BC00520=86202,981627,1075175
BC00521=81835,980250,1075175
BC00522=86350,984014,1075175
BC00523=118186,882849,1075175
BC00524=118313,879045,1075175
BC00525=118363,877523,1075175
BC00526=127351,877496,1075175
BC00527=127300,879018,1075175
BC00528=127173,882822,1075175
BC00529=149531,895732,1075175
BC00530=148249,891267,1075175
BC00531=148034,889482,1075175
BC00532=151775,889498,1075175
BC00533=152288,891284,1075175
BC00534=153569,895750,1075175
BC00535=119302,902119,1075175
BC00536=119440,897649,1075175
BC00537=119495,895861,1075175
BC00538=115974,895890,1075175
BC00539=115919,897678,1075175
BC00540=115781,902148,1075175
BC00541=206850,915693,1075175
BC00542=246637,921611,1075175
BC00543=251241,924622,1075175
BC00544=253082,925827,1075175
BC00545=305626,902567,1075175
BC00546=289523,905356,1075175
BC00547=289523,905356,1075175
BC00548=265997,901694,1075172
BC00549=265782,900020,1075175
BC00550=265246,895833,1075175
BC00551=152805,918674,1075175
BC00552=155644,922700,1075175
BC00553=156780,924310,1075175
BC00554=187141,913105,1075175
BC00555=135499,922155,1075175
BC00556=202417,924491,1075175
BC00557=204603,922909,1075175
BC00558=210067,918954,1075175
BC00559=285493,836258,1075175
BC00560=322674,778579,1075175
BC00561=322674,778579,1075175
BC00562=322674,778579,1075175
BC00563=322674,778579,1075175
BC00564=322674,778579,1075175
BC00565=322674,778579,1075175
BC00566=322674,778579,1075175
BC00567=322674,778579,1075175
BC00568=272555,769164,1075175
BC00569=266479,768023,1075175
BC00570=266479,768023,1075175
BC00571=267479,770239,1071365
BC00572=266799,769335,1075175
BC00573=266479,768023,1075175
BC00574=266479,768023,1075175
BC00575=266479,768023,1075175
BC00576=266479,768023,1075175
BC00577=235984,786404,1075175
BC00578=235984,786404,1075175
BC00579=235984,786404,1075175
BC00580=235984,786404,1075175
BC00581=235984,786404,1075175
BC00582=235984,786404,1075175
BC00583=235984,786404,1075175
BC00584=235984,786404,1075175
BC00585=237203,787368,1075175
BC00586=295022,827394,1075175
BC00587=205701,931185,1075175
BC00588=204812,932218,1075175
BC00589=205671,937629,1075175
BC00590=206015,939793,1075175
BC00591=202546,941762,1075175
BC00592=218293,952795,1075175
BC00593=218466,950486,1075175
BC00594=218898,944716,1075175
BC00595=188226,925402,1075175
BC00596=189298,932104,1075175
BC00597=189728,934784,1075175
BC00598=185375,937227,1075175
BC00599=184946,934546,1075175
BC00600=183874,927845,1075175
BC00601=163256,940528,1075175
BC00602=166760,944877,1075175
BC00603=168161,946617,1075175
BC00604=172960,943924,1075175
BC00605=171559,942185,1075175
BC00606=168055,937836,1075175
BC00607=205604,952176,1075175
BC00608=237375,964309,1075175
BC00609=234858,970014,1075175
BC00610=233851,972296,1075175
BC00611=237408,970622,1075175
BC00612=238426,968449,1075175
BC00613=241139,962660,1075175
BC00614=186195,958850,1075175
BC00615=137530,955476,1075175
BC00616=142340,959691,1075175
BC00617=135217,966057,1075175
BC00618=135217,966057,1075175
BC00619=134381,966543,1075175
BC00620=132263,964948,1075175
BC00621=126968,960962,1075175
BC00622=137530,955476,1075175
BC00623=284870,850327,1075175
BC00624=323104,941595,1075175
BC00625=324436,944989,1075175
BC00626=324969,946346,1075175
BC00627=379859,936839,1075175
BC00628=379326,935482,1075175
BC00629=377994,932088,1075175
BC00630=387025,925803,1075175
BC00631=391871,922431,1075175
BC00632=387133,926188,1075175
BC00633=385238,927691,1075175
BC00634=381091,925537,1075175
BC00635=365308,912570,1075175
BC00636=363166,908743,1075175
BC00637=364796,906869,1075175
BC00638=368870,902183,1075175
BC00639=358157,902408,1075175
BC00640=354876,908652,1075175
BC00641=353564,911150,1075175
BC00642=349138,907302,1075175
BC00643=357572,916934,1075175
BC00644=359178,914754,1075175
BC00645=363193,909304,1075175
BC00646=322758,853588,1075175
BC00647=135439,955204,1075175
BC00648=139952,957848,1075175
BC00649=141757,958906,1075175
BC00650=133040,997822,1075175
BC00651=133065,977483,1075175
BC00652=144047,1040883,1075175
BC00653=142698,1043050,1075175
BC00654=139327,1048468,1075175
BC00655=142698,1043050,1075175
BC00656=21214,672831,1075175
BC00657=48829,688840,1075175
BC00658=366911,902233,1075175
BC00659=366911,902233,1075175
BC00660=366911,902233,1075175
BC00661=366911,902233,1075175
BC00662=366911,902233,1075175
BC00663=366911,902233,1075175
BC00664=366911,902233,1075175
BC00665=366911,902233,1075175
BC00666=333056,895412,1075175
BC00667=333056,895412,1075175
BC00668=333056,895412,1075175
BC00669=333056,895412,1075175
BC00670=333056,895412,1075175
BC00671=333056,895412,1075175
BC00672=333056,895412,1075175
BC00673=333056,895412,1075175
BC00674=358091,902222,1075175
BC00675=358091,902222,1075175
BC00676=358091,902222,1075175
BC00677=358091,902222,1075175
BC00678=358091,902222,1075175
BC00679=358091,902222,1075175
BC00680=358091,902222,1075175
BC00681=358091,902222,1075175
BC00682=358091,902222,1075175
BC00683=358091,902222,1075175
BC00684=358091,902222,1075175
BC00685=358091,902222,1075175
BC00686=358091,902222,1075175
BC00687=358091,902222,1075175
BC00688=398174,894103,1075175
BC00689=398174,894103,1075175
BC00690=398174,894103,1075175
BC00691=398174,894103,1075175
BC00692=398174,894103,1075175
BC00693=398174,894103,1075175
BC00694=398174,894103,1075175
BC00695=398174,894103,1075175
BC00696=264903,781270,1075175
BC00697=264903,781270,1075175
BC00698=264904,781269,1075172
BC00699=264904,781269,1075171
BC00700=264904,781269,1075171
BC00701=264904,781269,1075168
BC00702=264904,781269,1075168
BC00703=264904,781269,1075168
BC00704=264904,781269,1075168
BC00705=264904,781269,1075168
BC00706=264904,781269,1075164
BC00707=264903,781270,1075175
BC00708=301264,775814,1075175
BC00709=301264,775814,1075175
BC00710=301264,775814,1075175
BC00711=301264,775814,1075175
BC00712=301264,775814,1075175
BC00713=301264,775814,1075175
BC00714=301264,775814,1075175
BC00715=301264,775814,1075175
BC00716=301264,775814,1075175
BC00717=301264,775814,1075175
BC00718=274235,786209,1075175
BC00719=238672,799885,1075175
BC00720=238672,799885,1075175
BC00721=238672,799885,1075175
BC00722=238672,799885,1075175
BC00723=238672,799885,1075175
BC00724=238672,799885,1075175
BC00725=238672,799885,1075175
BC00726=238672,799885,1075175
BC00727=238672,799884,1075171
BC00728=238672,799884,1075171
BC00729=238672,799885,1075175
BC00730=238672,799885,1075175
BC00731=238672,799885,1075175
BC00732=238672,799885,1075175
BC00733=318263,750454,1075175
BC00734=318263,750454,1075175
BC00735=318263,750454,1075175
BC00736=318263,750454,1075175
BC00737=318263,750454,1075175
BC00738=318263,750454,1075175
BC00739=318263,750454,1075175
BC00740=318263,750454,1075175
BC00741=318263,750454,1075175
BC00742=318263,750454,1075175
BC00743=318263,750454,1075175
BC00744=318263,750454,1075175
BC00745=318263,750454,1075175
BC00746=318263,750454,1075175
BC00747=318263,750454,1075175
BC00748=318263,750454,1075175
BC00749=318263,750454,1075175
BC00750=318263,750454,1075175
BC00751=318263,750454,1075175
BC00752=318263,750454,1075175
BC00753=318263,750454,1075175
BC00754=318263,750454,1075175
BC00755=318263,750454,1075175
BC00756=318263,750454,1075175
BC00757=318263,750454,1075175
BC00758=377114,750454,1075175
BC00759=397814,750454,1075175
BC00760=397814,750454,1075175
BC00761=397814,750454,1075175
BC00762=397814,750454,1075175
BC00763=397814,750454,1075175
BC00764=397814,750454,1075175
BC00765=397814,750454,1075175
BC00766=397814,750454,1075175
BC00767=397814,750454,1075175
BC00768=397814,750454,1075175
BC00769=397814,750454,1075175
BC00770=397814,750454,1075175
BC00771=397814,750454,1075175
BC00772=397814,750454,1075175
BC00773=397814,750454,1075175
BC00774=397814,750454,1075175
BC00775=397814,750454,1075175
BC00776=397814,750454,1075175
BC00777=397814,750454,1075175
BC00778=397814,750454,1075175
BC00779=383090,762961,1075175
BC00780=372387,772052,1075175
BC00781=296274,836703,1075175
BC00782=296274,836703,1075175
BC00783=296274,836703,1075175
BC00784=296274,836703,1075175
BC00785=296274,836703,1075175
BC00786=296274,836703,1075175
BC00787=296274,836703,1075175
BC00788=296274,836703,1075175
BC00789=296274,836703,1075175
BC00790=296274,836703,1075175
BC00791=296274,836703,1075175
BC00792=296274,836703,1075175
BC00793=296274,836703,1075175
BC00794=312215,899988,1075175
BC00795=312215,944285,1075175
BC00796=312215,944285,1075175
BC00797=312215,944285,1075175
BC00798=312215,944285,1075175
BC00799=312215,944285,1075175
BC00800=312215,944285,1075175
BC00801=312215,944285,1075175
BC00802=312215,944285,1075175
BC00803=312215,944285,1075175
BC00804=312215,944285,1075175
BC00805=312215,944285,1075175
BC00806=259299,938961,1075175
BC00807=259299,938961,1075175
BC00808=259299,938961,1075175
BC00809=259299,938961,1075175
BC00810=259299,938961,1075175
BC00811=259299,938961,1075175
BC00812=259299,938961,1075175
BC00813=259299,938961,1075175
BC00814=259299,938961,1075175
BC00815=259299,938961,1075175
BC00816=259299,938961,1075175
BC00817=259299,938961,1075175
BC00818=211531,951911,1075175
BC00819=211531,951911,1075175
BC00820=211531,951911,1075175
BC00821=211531,951911,1075175
BC00822=211531,951911,1075175
BC00823=211531,951911,1075175
BC00824=211531,951911,1075175
BC00825=211531,951911,1075175
BC00826=211531,951911,1075175
BC00827=211531,951911,1075175
BC00828=211531,951911,1075175
BC00829=182503,951872,1075175
BC00830=184369,953383,1075175
BC00831=184369,953399,1075175
BC00832=184333,953526,1075175
BC00833=184897,956550,1075175
BC00834=184333,953526,1075175
BC00835=184751,953664,1075175
BC00836=187887,953121,1075175
BC00837=184751,953664,1075175
BC00838=178222,948378,1075175
BC00839=171711,951911,1075175
BC00840=171711,959591,1075175
BC00841=171711,959591,1075175
BC00842=171711,959591,1075175
BC00843=171711,959591,1075175
BC00844=171711,959591,1075175
BC00845=171711,959591,1075175
BC00846=171711,959591,1075175
BC00847=171711,959591,1075175
BC00848=171711,959591,1075175
BC00849=182815,952263,1075175
BC00850=183711,957103,1075175
BC00851=184069,959047,1075174
BC00852=184070,959056,1075175
BC00853=184189,959079,1075175
BC00854=184752,962103,1075175
BC00855=184189,959079,1075175
BC00856=182935,952303,1075175
BC00857=182935,952303,1075175
BC00858=182935,952303,1075175
BC00859=123088,1061215,1075175
BC00860=126332,1055781,1075175
BC00861=127630,1053613,1075175
BC00862=127630,1053623,1075175
BC00863=127630,1053607,1075175
BC00864=153753,1064749,1075175
BC00865=152152,1062093,1075175
BC00866=153753,1064749,1075175
BC00867=104366,1038154,1075175
BC00868=107120,1036610,1075175
BC00869=104366,1038154,1075175
BC00870=97490,1044180,1075175
BC00871=121157,1044973,1075175
BC00872=140343,1045718,1075175
BC00873=158643,1046375,1075175
BC00874=155464,1041036,1075175
BC00875=155106,1040455,1075175
BC00876=155106,1040463,1075175
BC00877=155288,1040367,1075175
BC00878=153687,1037711,1075175
BC00879=155288,1040367,1075175
BC00880=158891,1046297,1075175
BC00881=211337,993614,1075175
BC00882=274623,983932,1075175
BC00883=371761,1043051,1075175
BC00884=331941,1063020,1075175
BC00885=331941,1063020,1075175
BC00886=331941,1063020,1075175
BC00887=331941,1063020,1075175
BC00888=331941,1063020,1075175
BC00889=331941,1063020,1075175
BC00890=331941,1063020,1075175
BC00891=331941,1063020,1075175
BC00892=331941,1063020,1075175
BC00893=331941,1063020,1075175
BC00894=331941,1063020,1075175
BC00895=331941,1063020,1075175
BC00896=331941,1063020,1075175
BC00897=371761,1043051,1075175
BC00898=371761,1043051,1075175
BC00899=371761,1043051,1075175
BC00900=371761,1043051,1075175
BC00901=371761,1043051,1075175
BC00902=371761,1043051,1075175
BC00903=371761,1043051,1075175
BC00904=371761,1043051,1075175
BC00905=371761,1043051,1075175
BC00906=371761,1043051,1075175
BC00907=371761,1043051,1075175
BC00908=371761,1043051,1075175
BC00909=371761,1043051,1075175
BC00910=371761,1043051,1075175
BC00911=371761,1043051,1075175
BC00912=314185,938855,1075175
BC00913=247671,970611,1075175
BC00914=247671,970611,1075175
BC00915=247671,970611,1075175
BC00916=247671,970611,1075175
BC00917=247671,970611,1075175
BC00918=247671,970611,1075175
BC00919=247671,970611,1075175
BC00920=247671,970611,1075175
BC00921=247671,970611,1075175
BC00922=247671,970611,1075175
BC00923=247671,970611,1075175
BC00924=247671,970611,1075175
BC00925=303037,872055,1075175
BC00926=380992,820655,1075175
BC00927=380992,820655,1075175
BC00928=380992,820655,1075175
BC00929=380992,820655,1075175
BC00930=380992,820655,1075175
BC00931=380992,820655,1075175
BC00932=380992,820655,1075175
BC00933=380992,820655,1075175
BC00934=380992,820655,1075175
BC00935=380992,820655,1075175
BC00936=380992,820655,1075175
BC00937=380992,820655,1075175
BC00938=275256,812324,1075175
BC00939=125716,897903,1075175
BC00940=125716,897903,1075175
BC00941=125716,897903,1075175
BC00942=125716,897903,1075175
BC00943=125716,897903,1075175
BC00944=125716,897903,1075174
BC00945=125716,897903,1075171
BC00946=125716,897903,1075175
BC00947=125716,897903,1075175
BC00948=125716,897903,1075175
BC00949=125716,897903,1075175
BC00950=125716,897903,1075175
BC00951=125716,897903,1075175
BC00952=325019,822543,1075229
BC00953=325019,822543,1075229
BC00954=325019,822543,1075229
BC00955=325019,822543,1075229
BC00956=325019,822543,1075229
BC00957=325019,822543,1075229
BC00958=325019,822543,1075229
BC00959=325019,822543,1075229
BC00960=325019,822543,1075229
BC00961=325019,822543,1075229
BC00962=325019,822543,1075229
BC00963=325019,822543,1075229
BC00964=240667,871930,1075210
BC00965=81335,965219,1075175
BC00966=81335,965219,1075175
BC00967=81335,965219,1075175
BC00968=81335,965219,1075175
BC00969=81335,965219,1075175
BC00970=81335,965219,1075175
BC00971=81335,965219,1075175
BC00972=81335,965219,1075175
BC00973=39891,972466,1075175
BC00974=39891,972466,1075175
BC00975=39891,972466,1075175
BC00976=39891,972466,1075175
BC00977=39891,972466,1075175
BC00978=39891,972466,1075175
BC00979=39891,972466,1075175
BC00980=39891,1005107,1075175
BC00981=39891,1005107,1075175
BC00982=39891,1005107,1075175
BC00983=39891,1005107,1075175
BC00984=39891,1005107,1075175
BC00985=39891,1005107,1075175
BC00986=39891,972466,1075175
BC00987=126064,942124,1075175
BC00988=145718,951183,1075175
BC00989=145718,951183,1075175
BC00990=145718,951183,1075175
BC00991=145718,951183,1075175
BC00992=145718,951183,1075175
BC00993=145718,951183,1075175
BC00994=145718,951183,1075175
BC00995=145718,951183,1075175
BC00996=145718,951183,1075175
BC00997=145718,951183,1075175
BC00998=145718,951183,1075175
BC00999=145718,951183,1075175
BC01000=127193,914007,1075175
BC01001=75497,867475,1075175
BC01002=75497,867475,1075175
BC01003=75497,867475,1075175
BC01004=75497,867475,1075175
BC01005=75497,867475,1075175
BC01006=75497,867475,1075175
BC01007=75497,867475,1075175
BC01008=75497,867475,1075175
BC01009=75497,867475,1075175
BC01010=75497,867475,1075175
BC01011=75497,867475,1075175
BC01012=75497,867475,1075175
BC01013=75497,867475,1075175
BC01014=75497,867475,1075175
BC01015=75497,867475,1075175
BC01016=75497,867475,1075175
BC01017=75497,867475,1075175
BC01018=58830,852413,1075175
BC01019=43274,838354,1075175
BC01020=43274,838354,1075175
BC01021=43274,838354,1075175
BC01022=43274,838354,1075175
BC01023=43274,838354,1075175
BC01024=43274,838354,1075175
BC01025=43274,838354,1075175
BC01026=43274,838354,1075175
BC01027=43274,838354,1075175
BC01028=191439,896290,1075175
BC01029=209593,874493,1075175
BC01030=209593,874493,1075175
BC01031=209593,874493,1075174
BC01032=209593,874493,1075171
BC01033=209593,874493,1075175
BC01034=209593,874493,1075175
BC01035=209216,850926,1075175
BC01036=226866,854473,1075175
BC01037=228835,855864,1075175
BC01038=228835,855864,1075175
BC01039=228834,855864,1075173
BC01040=228834,855864,1075173
BC01041=228835,855864,1075175
BC01042=228835,855864,1075175
BC01043=228835,855864,1075175
BC01044=228835,855864,1075175
BC01045=228835,855864,1075175
BC01046=212683,986357,1075175
BC01047=212683,1004517,1075175
BC01048=212247,999872,1075175
BC01049=212146,998778,1075171
BC01050=214955,996593,1075174
BC01051=222186,994128,1075175
BC01052=222622,998773,1075175
BC01053=293477,973063,1075175
BC01054=293477,973063,1075175
BC01055=293477,973063,1075175
BC01056=293477,973063,1075175
BC01057=293477,973063,1075175
BC01058=293477,973063,1075175
BC01059=293477,973063,1075175
BC01060=293477,973063,1075175
BC01061=248777,974412,1075175
BC01062=147624,1017934,1075175
BC01063=124950,1033375,1075175
BC01064=124950,1033375,1075175
BC01065=124950,1033375,1075175
BC01066=124950,1033375,1075174
BC01067=124950,1033375,1075175
BC01068=124950,1033375,1075175
BC01069=106678,1046165,1075175
BC01070=106678,1046165,1075175
BC01071=106678,1046165,1075175
BC01072=106678,1046165,1075175
BC01073=106678,1046165,1075175
BC01074=106678,1046165,1075175
BC01075=172863,1024486,1075175
BC01076=172427,1019841,1075175
BC01077=172326,1018747,1075171
BC01078=175135,1016562,1075174
BC01079=182366,1014097,1075175
BC01080=182802,1018742,1075175
BC01081=253657,993032,1075175
BC01082=253657,993032,1075175
BC01083=253657,993032,1075175
BC01084=253657,993032,1075175
BC01085=253657,993032,1075175
BC01086=253657,993032,1075175
BC01087=253657,993032,1075175
BC01088=253657,993032,1075175
BC01089=208957,994381,1075175
BC01090=107804,1037903,1075175
BC01091=85130,1053344,1075175
BC01092=85130,1053344,1075175
BC01093=85130,1053344,1075175
BC01094=85130,1053344,1075175
BC01095=85130,1053344,1075175
BC01096=85130,1053344,1075175
BC01097=66858,1066134,1075175
BC01098=66858,1066134,1075175
BC01099=66858,1066134,1075175
BC01100=66858,1066134,1075175
BC01101=66858,1066134,1075175
BC01102=66858,1066134,1075175
BC01103=106678,1034404,1075175
BC01104=288363,951317,1075175
BC01105=319880,932288,1075175
BC01106=316203,930177,1075175
BC01107=314732,929332,1075175
BC01108=314732,929332,1075175
BC01109=294141,940882,1075175
BC01110=285351,949486,1075175
BC01111=280844,953897,1075175
BC01112=254356,968931,1075172
BC01113=253996,970793,1075175
BC01114=256777,973747,1075175
BC01115=224914,994659,1075175
BC01116=193407,1014756,1075175
BC01117=196552,1009267,1075175
BC01118=197065,1008372,1075175
BC01119=197397,1007797,1075175
BC01120=196552,1009278,1075175
BC01121=193407,1014766,1075175
BC01122=170876,1031134,1075175
BC01123=153007,1044116,1075175
BC01124=153007,1044116,1075175
BC01125=155599,1038213,1075175
BC01126=156636,1035851,1075175
BC01127=230598,1025728,1075175
BC01128=222023,1030515,1075175
BC01129=222023,1030515,1075175
BC01130=118655,1062836,1075175
BC01131=118655,1062836,1075175
BC01132=118655,1062836,1075175
BC01133=176896,1055708,1075175
BC01134=225377,1010635,1075175
BC01135=228184,1010601,1075175
BC01136=235201,1010515,1075175
BC01137=242597,980334,1075175
BC01138=282680,816770,1075175
BC01139=287393,774165,1075175
BC01140=293866,776192,1075175
BC01141=296455,777002,1075175
BC01142=296337,777088,1075175
BC01143=296308,777110,1075175
BC01144=296189,777197,1075175
BC01145=293600,776386,1075175
BC01146=287127,774359,1075175
BC01147=265173,805126,1075175
BC01148=271841,806848,1075175
BC01149=274508,807537,1075175
BC01150=274508,807537,1075175
BC01151=271842,806893,1075175
BC01152=265174,805171,1075175
BC01153=347775,809657,1075175
BC01154=348436,809459,1075175
BC01155=348700,809380,1075175
BC01156=352833,807067,1075175
BC01157=364813,800347,1075175
BC01158=368942,798027,1075175
BC01159=368677,798106,1075175
BC01160=368016,798304,1075175
BC01161=368016,798304,1075175
BC01162=391344,687000,1075175
BC01163=391344,687000,1075175
BC01164=391344,687000,1075175
BC01165=391344,687000,1075175
BC01166=391344,687000,1075175
BC01167=391344,687000,1075175
BC01168=391344,687000,1075175
BC01169=391344,687000,1075175
BC01170=391344,687000,1075175
BC01171=391344,687000,1075175
BC01172=391344,687000,1075175
BC01173=391344,687000,1075175
BC01174=358873,687000,1075175
BC01175=250171,896024,1075175
BC01176=255370,893912,1075175
BC01177=257449,893067,1075174
BC01178=259851,897051,1075175
BC01179=270502,914711,1075175
BC01180=268422,915555,1075175
BC01181=263223,917668,1075175
BC01182=251695,824506,1075175
BC01183=253916,829548,1075175
BC01184=254804,831565,1075175
BC01185=231448,844598,1075175
BC01186=231448,844598,1075175
BC01187=189878,862044,1075175
BC01188=188570,860127,1075175
BC01189=185301,855336,1075175
BC01190=261332,833542,1075175
BC01191=297112,823286,1075175
BC01192=293523,829343,1075175
BC01193=292087,831765,1075175
BC01194=292088,831788,1075175
BC01195=293523,829365,1075175
BC01196=297112,823308,1075175
BC01197=297112,823286,1075175
BC01198=112345,954746,1075175
BC01199=112345,954746,1075175
BC01200=111546,959512,1075175
BC01201=111226,961418,1075175
BC01202=111226,961418,1075175
BC01203=111226,961418,1075175
BC01204=63698,969650,1075175
BC01205=63700,969637,1075175
BC01206=63700,969637,1075175
BC01207=63700,969637,1075175
BC01208=64817,962978,1075175
BC01209=55529,859309,1075175
BC01210=51595,858048,1075175
BC01211=50021,857544,1075175
BC01212=45895,833192,1075175
BC01213=46071,849801,1075175
BC01214=43912,844296,1075175
BC01215=45475,843733,1075175
BC01216=45475,843733,1075175
BC01217=45475,843733,1075175
BC01218=45475,843733,1075175
BC01219=45475,843733,1075175
BC01220=49382,842326,1075175
BC01221=32191,855540,1075175
BC01222=35199,856902,1075175
BC01223=36402,857447,1075175
BC01224=24170,872455,1075175
BC01225=24116,855865,1075175
BC01226=17601,856883,1075175
BC01227=10106,858388,1075175
BC01228=7107,859694,1075175
BC01229=124165,958731,1075175
BC01230=124477,964204,1075175
BC01231=124602,966393,1075175
BC01232=119899,967208,1075175
BC01233=114659,968116,1075175
BC01234=114534,965927,1075175
BC01235=114222,960453,1075175
BC01236=169497,963360,1075175
BC01237=218455,965934,1075175
BC01238=214431,967961,1075175
BC01239=212822,968772,1075175
BC01240=212822,968772,1075175
BC01241=212822,968772,1075175
BC01242=212822,968772,1075175
BC01243=218344,963319,1075175
BC01244=222368,961291,1075175
BC01245=147324,958268,1075175
BC01246=86350,984014,1075175
BC01247=90717,985390,1075175
BC01248=92241,985755,1075175
BC01249=87949,982178,1075175
BC01250=87949,982178,1075175
BC01251=87949,982178,1075175
BC01252=86202,981627,1075175
BC01253=81835,980250,1075175
BC01254=83182,969192,1075175
BC01255=84657,971884,1075175
BC01256=84782,974073,1075175
BC01257=80079,974888,1075175
BC01258=74839,975796,1075175
BC01259=74714,973607,1075175
BC01260=74402,968133,1075175
BC01261=129677,971040,1075175
BC01262=178635,973614,1075175
BC01263=174611,975641,1075175
BC01264=173002,976452,1075175
BC01265=173002,976452,1075175
BC01266=173002,976452,1075175
BC01267=173002,976452,1075175
BC01268=178524,970999,1075175
BC01269=182548,968971,1075175
BC01270=107504,965948,1075175
BC01271=46530,991694,1075175
BC01272=50897,993070,1075175
BC01273=52421,993435,1075175
BC01274=48129,989858,1075175
BC01275=48129,989858,1075175
BC01276=48129,989858,1075175
BC01277=46382,989307,1075175
BC01278=42015,987930,1075175
BC01279=86350,984014,1075175
BC01280=118186,882849,1075175
BC01281=118313,879045,1075175
BC01282=118363,877523,1075175
BC01283=127351,877496,1075175
BC01284=127300,879018,1075175
BC01285=127173,882822,1075175
BC01286=149531,895732,1075175
BC01287=148249,891267,1075175
BC01288=148034,889482,1075175
BC01289=151775,889498,1075175
BC01290=152288,891284,1075175
BC01291=153569,895750,1075175
BC01292=119302,902119,1075175
BC01293=119440,897649,1075175
BC01294=119495,895861,1075175
BC01295=115974,895890,1075175
BC01296=115919,897678,1075175
BC01297=115781,902148,1075175
BC01298=206850,915693,1075175
BC01299=246637,921611,1075175
BC01300=251241,924622,1075175
BC01301=253082,925827,1075175
BC01302=305626,902567,1075175
BC01303=289523,905356,1075175
BC01304=289523,905356,1075175
BC01305=265997,901694,1075172
BC01306=265782,900020,1075175
BC01307=265246,895833,1075175
BC01308=152805,918674,1075175
BC01309=155644,922700,1075175
BC01310=156780,924310,1075175
BC01311=187141,913105,1075175
BC01312=179441,914454,1075175
BC01313=179441,914454,1075175
BC01314=179441,914454,1075175
BC01315=120688,931609,1075175
BC01316=120688,931609,1036122
BC01317=120688,931609,1036122
BC01318=135499,922155,1075175
BC01319=196755,924293,1075175
BC01320=204603,922909,1075175
BC01321=210067,918954,1075175
BC01322=285493,836258,1075175
BC01323=322674,778579,1075175
BC01324=322674,778579,1075175
BC01325=322674,778579,1075175
BC01326=322674,778579,1075175
BC01327=322674,778579,1075175
BC01328=322674,778579,1075175
BC01329=322674,778579,1075175
BC01330=322674,778579,1075175
BC01331=272555,769164,1075175
BC01332=266479,768023,1075175
BC01333=266479,768023,1075175
BC01334=267479,770239,1071365
BC01335=266799,769335,1075175
BC01336=266479,768023,1075175
BC01337=266479,768023,1075175
BC01338=266479,768023,1075175
BC01339=266479,768023,1075175
BC01340=235984,786404,1075175
BC01341=235984,786404,1075175
BC01342=235984,786404,1075175
BC01343=235984,786404,1075175
BC01344=235984,786404,1075175
BC01345=235984,786404,1075175
BC01346=235984,786404,1075175
BC01347=235984,786404,1075175
BC01348=237203,787368,1075175
BC01349=295022,827394,1075175
BC01350=205701,931185,1075175
BC01351=204812,932218,1075175
BC01352=205671,937629,1075175
BC01353=206015,939793,1075175
BC01354=202546,941762,1075175
BC01355=218293,952795,1075175
BC01356=218466,950486,1075175
BC01357=218898,944716,1075175
BC01358=188226,925402,1075175
BC01359=189298,932104,1075175
BC01360=189728,934784,1075175
BC01361=185375,937227,1075175
BC01362=184946,934546,1075175
BC01363=183874,927845,1075175
BC01364=163256,940528,1075175
BC01365=166760,944877,1075175
BC01366=168161,946617,1075175
BC01367=172960,943924,1075175
BC01368=171559,942185,1075175
BC01369=168055,937836,1075175
BC01370=205604,952176,1075175
BC01371=237375,964309,1075175
BC01372=234858,970014,1075175
BC01373=233851,972296,1075175
BC01374=237408,970622,1075175
BC01375=238426,968449,1075175
BC01376=241139,962660,1075175
BC01377=186195,958850,1075175
BC01378=137530,955476,1075175
BC01379=142340,959691,1075175
BC01380=135217,966057,1075175
BC01381=135217,966057,1075175
BC01382=134381,966543,1075175
BC01383=132263,964948,1075175
BC01384=126968,960962,1075175
BC01385=137530,955476,1075175
BC01386=284870,850327,1075175
BC01387=323104,941595,1075175
BC01388=323297,942087,1075175
BC01389=323297,942087,1075175
BC01390=323297,942087,1075175
BC01391=324969,946346,1075175
BC01392=377020,937331,1075175
BC01393=379859,936839,1075175
BC01394=379326,935482,1075175
BC01395=377994,932088,1075175
BC01396=387025,925803,1075175
BC01397=391871,922431,1075175
BC01398=387133,926188,1075175
BC01399=385238,927691,1075175
BC01400=381091,925537,1075175
BC01401=365308,912570,1075175
BC01402=363166,908743,1075175
BC01403=364796,906869,1075175
BC01404=368870,902183,1075175
BC01405=358157,902408,1075175
BC01406=354876,908652,1075175
BC01407=353564,911150,1075175
BC01408=349138,907302,1075175
BC01409=357572,916934,1075175
BC01410=359178,914754,1075175
BC01411=363193,909304,1075175
BC01412=322758,853588,1075175
BC01413=135439,955204,1075175
BC01414=139952,957848,1075175
BC01415=141757,958906,1075175
BC01416=133040,997822,1075175
BC01417=133065,977483,1075175
BC01418=144047,1040883,1075175
BC01419=142698,1043050,1075175
BC01420=139327,1048468,1075175
BC01421=139327,1048468,1075175
BC01422=95619,955204,1075175
BC01423=100132,965528,1075175
BC01424=101937,966586,1075175
BC01425=93220,1005502,1075175
BC01426=93220,1005502,1075175
BC01427=93221,1030527,1075216
BC01428=93221,1030527,1075216
BC01429=99566,1045795,1075190
BC01430=142698,1043050,1075175
BC01431=206177,1018673,1075175
BC01432=252443,1048931,1075175
BC01433=258757,1029159,1075175
BC01434=290253,930536,1075175
BC01435=290253,930536,1075175
BC01436=290253,930536,1075175
BC01437=297151,966120,1075172
BC01438=297151,997903,1075172
BC01439=297151,997903,1075172
BC01440=297194,1021413,1075172
BC01441=297194,1021413,1075172
BC01442=21214,672831,1075175
BC01443=21214,672831,429902
BC01444=66815,724118,419761
BC01445=110240,772957,337669
BC01446=124996,789553,122283
BC01447=124996,789553,122283
BC01448=124996,789553,122283
BC01449=124996,789553,122283
BC01450=124996,789553,122283
BC01451=124996,789553,122283
BC01452=124996,789553,122283
BC01453=124996,789553,122283
BC01454=124996,789553,122283
BC01455=124996,789553,122283
BC01456=124996,789553,122283
BC01457=124996,789553,122283
BC01458=124996,789553,122283
BC01459=124996,789553,122283
BC01460=124996,789553,122283
BC01461=136729,789553,283981
BC01462=136729,789553,283981
BC01463=136729,789553,283981
BC01464=136729,789553,283981
BC01465=136729,789553,283981
BC01466=136729,789553,283981
BC01467=136729,789553,283981
BC01468=136729,789553,283981
BC01469=136729,789553,283981
BC01470=136729,789553,283981
BC01471=163194,789553,386705
BC01472=163194,789553,386705
BC01473=163194,789553,386705
BC01474=163194,789553,386705
BC01475=163194,789553,386705
BC01476=163194,789553,386705
BC01477=163194,789553,386705
BC01478=163194,789553,386705
BC01479=163194,789553,386705
BC01480=163194,789553,386705
BC01481=110240,772957,337669
BC01482=66815,724118,419761
BC01483=66815,670858,419761
BC01484=252765,670858,277331
BC01485=322808,760288,131711
BC01486=322808,760288,131711
BC01487=322808,760288,131711
BC01488=322808,760288,131711
BC01489=322808,760288,131711
BC01490=322808,760288,131711
BC01491=322808,760288,131711
BC01492=322808,760288,131711
BC01493=322808,760288,131711
BC01494=335534,789553,204922
BC01495=335534,789553,204922
BC01496=335534,789553,204922
BC01497=335534,789553,204922
BC01498=335534,789553,204922
BC01499=335534,789553,204922
BC01500=335534,789553,204922
BC01501=335534,789553,204922
BC01502=335534,789553,204922
BC01503=335534,789553,204922
BC01504=335534,789553,204922
BC01505=335534,789553,204922
BC01506=335534,789553,204922
BC01507=335534,789553,204922
BC01508=335534,789553,204922
BC01509=335534,789553,204922
BC01510=344006,752651,139062
BC01511=344006,752651,139062
BC01512=344005,752652,139060
BC01513=344005,752652,139060
BC01514=344005,752652,139060
BC01515=344005,752652,139060
BC01516=344005,752652,139060
BC01517=344005,752652,139060
BC01518=344005,752652,139060
BC01519=344005,752652,139060
BC01520=344005,752652,139060
BC01521=344005,752652,139060
BC01522=344005,752652,139060
BC01523=344005,752652,139060
BC01524=344005,752652,139060
BC01525=344006,752651,139062
BC01526=300933,750795,218908
BC01527=283893,750061,250495
BC01528=276320,749735,264534
BC01529=276320,749735,264534
BC01530=276320,749735,264534
BC01531=276320,749735,264532
BC01532=276320,749735,264532
BC01533=276320,749735,264532
BC01534=276320,749735,264532
BC01535=276320,749735,264532
BC01536=276320,749735,264532
BC01537=276320,749735,264532
BC01538=276320,749735,264532
BC01539=276320,749736,264531
BC01540=276320,749736,264531
BC01541=276320,749736,264531
BC01542=276320,749736,264531
BC01543=276320,749735,264534
BC01544=248857,763770,138691
BC01545=248857,763770,138691
BC01546=248857,763770,138691
BC01547=248857,763770,138691
BC01548=248857,763770,138691
BC01549=248857,763770,138691
BC01550=248857,763770,138691
BC01551=248857,763770,138691
BC01552=248857,763770,138691
BC01553=248857,763770,138691
BC01554=248857,763770,138691
BC01555=248857,763770,138691
BC01556=248857,763770,138691
BC01557=248857,763770,138691
BC01558=248857,763770,138691
BC01559=248857,763770,138691
BC01560=287864,789553,132710
BC01561=287864,789553,132710
BC01562=287864,789553,132710
BC01563=287864,789553,132710
BC01564=287864,789553,132710
BC01565=287864,789553,132710
BC01566=287864,789553,132710
BC01567=287864,789553,132710
BC01568=287864,789553,132710
BC01569=287864,789553,132710
BC01570=287864,789553,132710
BC01571=287864,789553,132710
BC01572=279829,789553,53
BC01573=279829,789553,53
BC01574=279829,789553,53
BC01575=279829,789553,53
BC01576=279829,789553,53
BC01577=279829,789553,53
BC01578=279829,789553,53
BC01579=279829,789553,53
BC01580=279829,789553,53
BC01581=279829,789553,53
BC01582=279829,789553,53
BC01583=279829,789553,53
BC01584=279829,789553,53
BC01585=312324,789553,158805
BC01586=312324,789553,158805
BC01587=312324,789553,158804
BC01588=312324,789553,158805
BC01589=312324,789553,158805
BC01590=312324,789553,158805
BC01591=303082,768394,105099
BC01592=303082,768394,105099
BC01593=303082,768394,105099
BC01594=303082,768394,105099
BC01595=303082,768394,105099
BC01596=303082,768394,105099
BC01597=287868,781442,183325
BC01598=278410,789553,231953
BC01599=278410,789553,231953
BC01600=278410,789553,231953
BC01601=278410,789553,231953
BC01602=278410,789553,231953
BC01603=278410,789553,231953
BC01604=283893,750061,250495
BC01605=300933,750795,218908
BC01606=376723,772526,120737
BC01607=376723,772526,120737
BC01608=376723,772526,120737
BC01609=376723,772526,120737
BC01610=376723,772526,120737
BC01611=376723,772526,120737
BC01612=385013,737075,95404
BC01613=385013,737075,95404
BC01614=385013,737075,95404
BC01615=385013,737075,95404
BC01616=385013,737075,95404
BC01617=385013,737075,95404
BC01618=365962,760163,122379
BC01619=365962,760163,122379
BC01620=365962,760163,122379
BC01621=365962,760163,122379
BC01622=365962,760163,122379
BC01623=365962,760163,122379
BC01624=365962,760163,122379
BC01625=252765,670858,277331
BC01626=66815,670858,419761
BC01627=66815,724118,419761
BC01628=110240,772957,337669
BC01629=118803,789553,240458
BC01630=118803,789553,240458
BC01631=118803,789553,240458
BC01632=118803,789553,240458
BC01633=118803,789553,240458
BC01634=118803,789553,240458
BC01635=130259,789553,198376
BC01636=110709,789553,198376
BC01637=113251,789553,198376
BC01638=113251,789553,198376
BC01639=113251,789553,198376
BC01640=113251,789553,198376
BC01641=113251,789553,198376
BC01642=113251,789553,198376
BC01643=113251,789553,198376
BC01644=113251,789553,198376
BC01645=113251,789553,198376
BC01646=113251,789553,198376
BC01647=113251,789553,198376
BC01648=113251,789553,198376
BC01649=113251,789553,198376
BC01650=113251,789553,228042
BC01651=113251,789553,280292
BC01652=113251,789553,280290
BC01653=113251,789553,280290
BC01654=113251,789553,280290
BC01655=113251,789553,280290
BC01656=113251,789553,280290
BC01657=113251,789553,280290
BC01658=113251,789553,280290
BC01659=110240,772957,337669
BC01660=66815,724118,419761
BC01661=66815,670858,419761
BC01662=252765,670858,277331
BC01663=298333,782774,240815
BC01664=298333,782774,240815
BC01665=298333,782774,240815
BC01666=298333,782774,240815
BC01667=298333,782774,240815
BC01668=298333,782774,240815
BC01669=277596,773081,190929
BC01670=277596,773081,190929
BC01671=277596,773081,190929
BC01672=277596,773081,190929
BC01673=277596,773081,190929
BC01674=277596,773081,190929
BC01675=252765,670858,277331
BC01676=66815,670858,419761
BC01677=66815,724118,419761
BC01678=110240,772957,337669
BC01679=116545,789553,319269
BC01680=116545,789553,319269
BC01681=116545,789553,319269
BC01682=116545,789553,319269
BC01683=116545,789553,319269
BC01684=116545,789553,319269
BC01685=104258,789553,379308
BC01686=104258,789553,379308
BC01687=104258,789553,379308
BC01688=104258,789553,379308
BC01689=104258,789553,379308
BC01690=104258,789553,379308
BC01691=110240,772957,337669
BC01692=66815,724118,419761
BC01693=66815,670858,419761
BC01694=252765,670858,277331
BC01695=286674,787255,240962
BC01696=286675,787255,240962
BC01697=286675,787255,240962
BC01698=286675,787255,240962
BC01699=286674,787255,240962
BC01700=286674,787255,240962
BC01701=267109,758037,158941
BC01702=267109,758037,158941
BC01703=267109,758037,158941
BC01704=267109,758037,158941
BC01705=267109,758037,158941
BC01706=267109,758037,158941
BC01707=283893,750061,250495
BC01708=360336,760725,110934
BC01709=360336,760725,110934
BC01710=360336,760725,110934
BC01711=360336,760725,110934
BC01712=360336,760725,110934
BC01713=360336,760725,110934
BC01714=371149,789553,191296
BC01715=371149,789553,191296
BC01716=371149,789553,191296
BC01717=371149,789553,191296
BC01718=371149,789553,191296
BC01719=371149,789553,191296
BC01720=283893,750061,250495
BC01721=292970,789553,136523
BC01722=292970,789553,136523
BC01723=292970,789553,136523
BC01724=292970,789553,136523
BC01725=292970,789553,136523
BC01726=292970,789552,136519
BC01727=292970,789553,136523
BC01728=292970,789553,136523
BC01729=256495,759418,21571
BC01730=256495,759418,21571
BC01731=256495,759418,21571
BC01732=256495,759418,21571
BC01733=256495,759418,21571
BC01734=256495,759418,21571
BC01735=256075,748610,41729
BC01736=255916,738170,60084
BC01737=255916,738170,60084
BC01738=255916,738170,60084
BC01739=255916,738170,60084
BC01740=255916,738170,60084
BC01741=255916,738170,60084
BC01742=262339,748900,193466
BC01743=165820,667836,534036
BC01744=21214,672831,1075175
EC00000=798156,1112951
EC00001=798156,1112951
EC00002=798156,1112951
EC00003=798156,1112951
EC00004=798156,1112951
EC00005=798156,1112951
EC00006=798156,1112951
EC00007=798156,1112951
EC00008=798156,1112951
EC00009=798156,1112951
EC00010=798156,1112951
EC00011=798156,1112951
EC00012=798156,1112951
EC00013=798156,1112951
EC00014=798156,1112951
EC00015=798156,1112951
EC00016=798156,1112951
EC00017=798156,1112951
EC00018=798156,1112951
EC00019=798156,1112951
EC00020=798156,1112951
EC00021=798156,1112951
EC00022=798156,1112951
EC00023=798156,1112951
EC00024=798156,1112951
EC00025=798156,1112951
EC00026=798156,1112951
EC00027=798156,1112951
EC00028=798156,1112951
EC00029=798156,1112951
EC00030=798156,1112951
EC00031=798156,1112951
EC00032=798156,1112951
EC00033=798156,1112951
EC00034=798156,1112951
EC00035=798155,1112950
EC00036=798155,1112950
EC00037=798155,1112950
EC00038=798154,1112949
EC00039=798154,1112949
EC00040=798154,1112949
EC00041=798154,1112949
EC00042=798154,1112949
EC00043=798153,1112949
EC00044=798156,1112951
EC00045=798156,1112951
EC00046=798156,1112951
EC00047=798156,1112951
EC00048=798156,1112951
EC00049=798156,1112951
EC00050=798156,1112951
EC00051=798156,1112951
EC00052=798156,1112951
EC00053=798156,1112951
EC00054=798156,1112951
EC00055=798156,1112951
EC00056=798156,1112951
EC00057=798156,1112951
EC00058=798156,1112951
EC00059=798156,1112951
EC00060=798156,1112951
EC00061=798156,1112951
EC00062=798156,1112951
EC00063=798156,1112951
EC00064=798155,1112950
EC00065=798155,1112950
EC00066=798156,1112951
EC00067=798156,1112951
EC00068=798156,1112951
EC00069=798156,1112951
EC00070=798156,1112951
EC00071=798156,1112951
EC00072=798156,1112951
EC00073=798156,1112951
EC00074=798156,1112951
EC00075=798156,1112951
EC00076=798156,1112951
EC00077=798156,1112951
EC00078=798156,1112951
EC00079=798156,1112951
EC00080=798156,1112951
EC00081=798156,1112951
EC00082=798156,1112951
EC00083=798156,1112951
EC00084=798156,1112951
EC00085=798156,1112951
EC00086=798156,1112951
EC00087=798156,1112951
EC00088=798156,1112951
EC00089=798156,1112951
EC00090=798156,1112951
EC00091=798156,1112951
EC00092=798156,1112951
EC00093=798156,1112951
EC00094=798156,1112951
EC00095=798156,1112951
EC00096=798156,1112951
EC00097=798156,1112951
EC00098=798156,1112951
EC00099=798156,1112951
EC00100=798156,1112951
EC00101=798156,1112951
EC00102=798156,1112951
EC00103=798156,1112951
EC00104=798156,1112951
EC00105=798156,1112951
EC00106=798156,1112951
EC00107=798156,1112951
EC00108=798156,1112951
EC00109=798156,1112951
EC00110=798156,1112951
EC00111=798156,1112951
EC00112=798156,1112951
EC00113=798156,1112951
EC00114=798156,1112951
EC00115=798156,1112951
EC00116=798156,1112951
EC00117=798156,1112951
EC00118=798156,1112951
EC00119=798156,1112951
EC00120=798156,1112951
EC00121=798156,1112951
EC00122=798156,1112951
EC00123=798156,1112951
EC00124=798156,1112951
EC00125=798156,1112951
EC00126=798156,1112951
EC00127=798156,1112951
EC00128=798156,1112951
EC00129=798156,1112951
EC00130=798156,1112951
EC00131=798156,1112951
EC00132=798156,1112951
EC00133=798156,1112951
EC00134=798156,1112951
EC00135=798156,1112951
EC00136=798156,1112951
EC00137=798156,1112951
EC00138=798156,1112951
EC00139=798156,1112951
EC00140=798156,1112951
EC00141=798156,1112951
EC00142=798156,1112951
EC00143=798156,1112951
EC00144=798156,1112951
EC00145=798156,1112951
EC00146=798156,1112951
EC00147=798156,1112951
EC00148=798156,1112951
EC00149=798156,1112951
EC00150=798156,1112951
EC00151=798156,1112951
EC00152=798156,1112951
EC00153=798156,1112951
EC00154=798156,1112951
EC00155=798156,1112951
EC00156=798156,1112951
EC00157=798156,1112951
EC00158=798156,1112951
EC00159=798156,1112951
EC00160=798156,1112951
EC00161=798156,1112951
EC00162=798156,1112951
EC00163=798156,1112951
EC00164=798156,1112951
EC00165=798156,1112951
EC00166=798156,1112951
EC00167=798156,1112951
EC00168=798156,1112951
EC00169=798156,1112951
EC00170=798156,1112951
EC00171=798156,1112951
EC00172=798156,1112951
EC00173=798156,1112951
EC00174=798156,1112951
EC00175=798156,1112951
EC00176=798156,1112951
EC00177=798156,1112951
EC00178=798155,1112950
EC00179=798156,1112951
EC00180=798156,1112951
EC00181=798156,1112951
EC00182=798156,1112951
EC00183=798156,1112951
EC00184=798156,1112951
EC00185=798156,1112951
EC00186=798156,1112951
EC00187=798156,1112951
EC00188=798156,1112951
EC00189=798156,1112951
EC00190=798156,1112951
EC00191=798156,1112951
EC00192=798156,1112951
EC00193=798156,1112951
EC00194=798156,1112951
EC00195=798156,1112951
EC00196=798156,1112951
EC00197=798156,1112951
EC00198=798156,1112951
EC00199=798156,1112951
EC00200=798156,1112951
EC00201=798156,1112951
EC00202=798156,1112951
EC00203=798156,1112951
EC00204=798156,1112951
EC00205=798156,1112951
EC00206=798156,1112951
EC00207=798156,1112951
EC00208=798156,1112951
EC00209=798156,1112951
EC00210=798156,1112951
EC00211=798156,1112951
EC00212=798156,1112951
EC00213=798156,1112951
EC00214=798156,1112951
EC00215=798156,1112951
EC00216=798156,1112951
EC00217=798156,1112951
EC00218=798156,1112951
EC00219=798156,1112951
EC00220=798156,1112951
EC00221=798156,1112951
EC00222=798156,1112951
EC00223=798156,1112951
EC00224=798156,1112951
EC00225=798156,1112951
EC00226=798156,1112951
EC00227=798156,1112951
EC00228=798156,1112951
EC00229=798156,1112951
EC00230=798156,1112951
EC00231=798156,1112951
EC00232=798156,1112951
EC00233=798156,1112951
EC00234=798156,1112951
EC00235=798156,1112951
EC00236=798156,1112951
EC00237=798156,1112951
EC00238=798156,1112951
EC00239=798156,1112951
EC00240=798156,1112951
EC00241=798156,1112951
EC00242=798156,1112951
EC00243=798156,1112951
EC00244=798156,1112951
EC00245=798156,1112951
EC00246=798156,1112951
EC00247=798156,1112951
EC00248=798156,1112951
EC00249=798156,1112951
EC00250=798156,1112951
EC00251=798156,1112951
EC00252=798156,1112951
EC00253=798156,1112951
EC00254=798156,1112951
EC00255=798156,1112951
EC00256=798155,1112951
EC00257=798156,1112951
EC00258=798156,1112951
EC00259=798156,1112951
EC00260=798156,1112951
EC00261=798156,1112951
EC00262=798156,1112951
EC00263=798156,1112951
EC00264=798156,1112951
EC00265=798156,1112951
EC00266=798156,1112951
EC00267=798156,1112951
EC00268=798156,1112951
EC00269=798156,1112951
EC00270=798156,1112951
EC00271=798156,1112951
EC00272=798156,1112951
EC00273=798156,1112951
EC00274=798156,1112951
EC00275=798156,1112951
EC00276=798156,1112951
EC00277=798156,1112951
EC00278=798156,1112951
EC00279=798156,1112951
EC00280=798156,1112951
EC00281=798156,1112951
EC00282=798156,1112951
EC00283=798156,1112951
EC00284=798156,1112951
EC00285=798156,1112951
EC00286=798156,1112951
EC00287=798156,1112951
EC00288=798156,1112951
EC00289=798156,1112951
EC00290=798156,1112951
EC00291=798156,1112951
EC00292=798156,1112951
EC00293=798156,1112951
EC00294=798156,1112951
EC00295=798156,1112951
EC00296=798156,1112951
EC00297=798156,1112951
EC00298=798156,1112951
EC00299=798156,1112951
EC00300=798156,1112951
EC00301=798156,1112951
EC00302=798156,1112951
EC00303=798156,1112951
EC00304=798156,1112951
EC00305=798156,1112951
EC00306=798156,1112951
EC00307=798156,1112951
EC00308=798156,1112951
EC00309=798156,1112951
EC00310=798156,1112951
EC00311=798156,1112951
EC00312=798156,1112951
EC00313=798156,1112951
EC00314=798156,1112951
EC00315=798156,1112951
EC00316=798156,1112951
EC00317=798156,1112951
EC00318=798156,1112951
EC00319=798156,1112951
EC00320=798156,1112951
EC00321=798156,1112951
EC00322=798156,1112951
EC00323=798156,1112951
EC00324=798156,1112951
EC00325=798156,1112951
EC00326=798156,1112951
EC00327=798156,1112951
EC00328=798156,1112951
EC00329=798156,1112951
EC00330=798156,1112951
EC00331=798156,1112951
EC00332=798156,1112951
EC00333=798156,1112951
EC00334=798156,1112951
EC00335=798156,1112951
EC00336=798156,1112951
EC00337=798155,1112950
EC00338=798156,1112951
EC00339=798156,1112951
EC00340=798156,1112951
EC00341=798156,1112951
EC00342=798156,1112951
EC00343=798156,1112951
EC00344=798155,1112951
EC00345=798155,1112951
EC00346=798156,1112951
EC00347=798156,1112951
EC00348=798156,1112951
EC00349=798156,1112951
EC00350=798156,1112951
EC00351=798156,1112951
EC00352=798156,1112951
EC00353=798156,1112951
EC00354=798155,1112950
EC00355=798156,1112951
EC00356=798156,1112951
EC00357=798156,1112951
EC00358=798156,1112951
EC00359=798156,1112951
EC00360=798156,1112951
EC00361=798156,1112951
EC00362=798156,1112951
EC00363=798156,1112951
EC00364=798156,1112951
EC00365=798156,1112951
EC00366=798156,1112951
EC00367=798156,1112951
EC00368=798156,1112951
EC00369=798156,1112951
EC00370=798156,1112951
EC00371=798156,1112951
EC00372=798156,1112951
EC00373=798156,1112951
EC00374=798156,1112951
EC00375=798156,1112951
EC00376=798156,1112951
EC00377=798156,1112951
EC00378=798156,1112951
EC00379=798156,1112951
EC00380=798156,1112951
EC00381=798156,1112951
EC00382=798156,1112951
EC00383=798156,1112951
EC00384=798156,1112951
EC00385=798156,1112951
EC00386=798156,1112951
EC00387=798156,1112951
EC00388=798156,1112951
EC00389=798155,1112950
EC00390=798156,1112951
EC00391=798156,1112951
EC00392=798156,1112951
EC00393=798156,1112951
EC00394=798156,1112951
EC00395=798156,1112951
EC00396=798156,1112951
EC00397=798156,1112951
EC00398=798156,1112951
EC00399=798156,1112951
EC00400=798156,1112951
EC00401=798156,1112951
EC00402=798156,1112951
EC00403=798156,1112951
EC00404=798156,1112951
EC00405=798156,1112951
EC00406=798156,1112951
EC00407=798156,1112951
EC00408=798156,1112951
EC00409=798156,1112951
EC00410=798156,1112951
EC00411=798156,1112951
EC00412=798156,1112951
EC00413=798156,1112951
EC00414=798156,1112951
EC00415=798156,1112951
EC00416=798156,1112951
EC00417=798156,1112951
EC00418=798156,1112951
EC00419=798156,1112951
EC00420=798156,1112951
EC00421=798156,1112951
EC00422=798156,1112951
EC00423=798156,1112951
EC00424=798156,1112951
EC00425=798156,1112951
EC00426=798156,1112951
EC00427=798156,1112951
EC00428=798156,1112951
EC00429=798156,1112951
EC00430=798156,1112951
EC00431=798156,1112951
EC00432=798156,1112951
EC00433=798156,1112951
EC00434=798156,1112951
EC00435=798156,1112951
EC00436=798156,1112951
EC00437=798156,1112951
EC00438=798156,1112951
EC00439=798156,1112951
EC00440=798156,1112951
EC00441=798156,1112951
EC00442=798156,1112951
EC00443=798156,1112951
EC00444=798156,1112951
EC00445=798156,1112951
EC00446=798156,1112951
EC00447=798156,1112951
EC00448=798156,1112951
EC00449=798156,1112951
EC00450=798156,1112951
EC00451=798156,1112951
EC00452=798156,1112951
EC00453=798156,1112951
EC00454=798156,1112951
EC00455=798156,1112951
EC00456=798156,1112951
EC00457=798156,1112951
EC00458=798156,1112951
EC00459=798156,1112951
EC00460=798156,1112951
EC00461=798156,1112951
EC00462=798156,1112951
EC00463=798156,1112951
EC00464=798156,1112951
EC00465=798156,1112951
EC00466=798156,1112951
EC00467=798156,1112951
EC00468=798156,1112951
EC00469=798156,1112951
EC00470=798156,1112951
EC00471=798156,1112951
EC00472=798156,1112951
EC00473=798156,1112951
EC00474=798156,1112951
EC00475=798156,1112951
EC00476=798156,1112951
EC00477=798156,1112951
EC00478=798156,1112951
EC00479=798156,1112951
EC00480=798156,1112951
EC00481=798156,1112951
EC00482=798156,1112951
EC00483=798156,1112951
EC00484=798156,1112951
EC00485=798156,1112951
EC00486=798156,1112951
EC00487=798156,1112951
EC00488=798156,1112951
EC00489=798156,1112951
EC00490=798156,1112951
EC00491=798156,1112951
EC00492=798156,1112951
EC00493=798156,1112951
EC00494=798156,1112951
EC00495=798156,1112951
EC00496=798156,1112951
EC00497=798156,1112951
EC00498=798156,1112951
EC00499=798156,1112951
EC00500=798156,1112951
EC00501=798156,1112951
EC00502=798156,1112951
EC00503=798156,1112951
EC00504=798156,1112951
EC00505=798156,1112951
EC00506=798156,1112951
EC00507=798156,1112951
EC00508=798156,1112951
EC00509=798156,1112951
EC00510=798156,1112951
EC00511=798156,1112951
EC00512=798156,1112951
EC00513=798156,1112951
EC00514=798156,1112951
EC00515=798156,1112951
EC00516=798156,1112951
EC00517=798156,1112951
EC00518=798156,1112951
EC00519=798156,1112951
EC00520=798156,1112951
EC00521=798156,1112951
EC00522=798156,1112951
EC00523=798156,1112951
EC00524=798156,1112951
EC00525=798156,1112951
EC00526=798156,1112951
EC00527=798156,1112951
EC00528=798156,1112951
EC00529=798156,1112951
EC00530=798156,1112951
EC00531=798156,1112951
EC00532=798156,1112951
EC00533=798156,1112951
EC00534=798156,1112951
EC00535=798156,1112951
EC00536=798156,1112951
EC00537=798156,1112951
EC00538=798156,1112951
EC00539=798156,1112951
EC00540=798156,1112951
EC00541=798156,1112951
EC00542=798156,1112951
EC00543=798156,1112951
EC00544=798156,1112951
EC00545=798156,1112951
EC00546=798156,1112951
EC00547=798156,1112951
EC00548=798155,1112950
EC00549=798156,1112951
EC00550=798156,1112951
EC00551=798156,1112951
EC00552=798156,1112951
EC00553=798156,1112951
EC00554=798156,1112951
EC00555=798156,1112951
EC00556=798156,1112951
EC00557=798156,1112951
EC00558=798156,1112951
EC00559=798156,1112951
EC00560=798156,1112951
EC00561=798156,1112951
EC00562=798156,1112951
EC00563=798156,1112951
EC00564=798156,1112951
EC00565=798156,1112951
EC00566=798156,1112951
EC00567=798156,1112951
EC00568=798156,1112951
EC00569=798156,1112951
EC00570=798156,1112951
EC00571=798156,1112951
EC00572=798156,1112951
EC00573=798156,1112951
EC00574=798156,1112951
EC00575=798156,1112951
EC00576=798156,1112951
EC00577=798156,1112951
EC00578=798156,1112951
EC00579=798156,1112951
EC00580=798156,1112951
EC00581=798156,1112951
EC00582=798156,1112951
EC00583=798156,1112951
EC00584=798156,1112951
EC00585=798156,1112951
EC00586=798156,1112951
EC00587=798156,1112951
EC00588=798156,1112951
EC00589=798156,1112951
EC00590=798156,1112951
EC00591=798156,1112951
EC00592=798156,1112951
EC00593=798156,1112951
EC00594=798156,1112951
EC00595=798156,1112951
EC00596=798156,1112951
EC00597=798156,1112951
EC00598=798156,1112951
EC00599=798156,1112951
EC00600=798156,1112951
EC00601=798156,1112951
EC00602=798156,1112951
EC00603=798156,1112951
EC00604=798156,1112951
EC00605=798156,1112951
EC00606=798156,1112951
EC00607=798156,1112951
EC00608=798156,1112951
EC00609=798156,1112951
EC00610=798156,1112951
EC00611=798156,1112951
EC00612=798156,1112951
EC00613=798156,1112951
EC00614=798156,1112951
EC00615=798156,1112951
EC00616=798156,1112951
EC00617=798156,1112951
EC00618=798156,1112951
EC00619=798156,1112951
EC00620=798156,1112951
EC00621=798156,1112951
EC00622=798156,1112951
EC00623=798156,1112951
EC00624=798156,1112951
EC00625=798156,1112951
EC00626=798156,1112951
EC00627=798156,1112951
EC00628=798156,1112951
EC00629=798156,1112951
EC00630=798156,1112951
EC00631=798156,1112951
EC00632=798156,1112951
EC00633=798156,1112951
EC00634=798156,1112951
EC00635=798156,1112951
EC00636=798156,1112951
EC00637=798156,1112951
EC00638=798156,1112951
EC00639=798156,1112951
EC00640=798156,1112951
EC00641=798156,1112951
EC00642=798156,1112951
EC00643=798156,1112951
EC00644=798156,1112951
EC00645=798156,1112951
EC00646=798156,1112951
EC00647=798156,1112951
EC00648=798156,1112951
EC00649=798156,1112951
EC00650=798156,1112951
EC00651=798156,1112951
EC00652=798156,1112951
EC00653=798156,1112951
EC00654=798156,1112951
EC00655=798156,1112951
EC00656=798156,1112951
EC00657=798156,1112951
EC00658=798156,1112951
EC00659=798156,1112951
EC00660=798156,1112951
EC00661=798156,1112951
EC00662=798156,1112951
EC00663=798156,1112951
EC00664=798156,1112951
EC00665=798156,1112951
EC00666=798156,1112951
EC00667=798156,1112951
EC00668=798156,1112951
EC00669=798156,1112951
EC00670=798156,1112951
EC00671=798156,1112951
EC00672=798156,1112951
EC00673=798156,1112951
EC00674=798156,1112951
EC00675=798156,1112951
EC00676=798156,1112951
EC00677=798156,1112951
EC00678=798156,1112951
EC00679=798156,1112951
EC00680=798156,1112951
EC00681=798156,1112951
EC00682=798156,1112951
EC00683=798156,1112951
EC00684=798156,1112951
EC00685=798156,1112951
EC00686=798156,1112951
EC00687=798156,1112951
EC00688=798156,1112951
EC00689=798156,1112951
EC00690=798156,1112951
EC00691=798156,1112951
EC00692=798156,1112951
EC00693=798156,1112951
EC00694=798156,1112951
EC00695=798156,1112951
EC00696=798156,1112951
EC00697=798156,1112951
EC00698=798155,1112950
EC00699=798155,1112950
EC00700=798155,1112950
EC00701=798154,1112949
EC00702=798154,1112949
EC00703=798154,1112949
EC00704=798154,1112949
EC00705=798154,1112949
EC00706=798153,1112949
EC00707=798156,1112951
EC00708=798156,1112951
EC00709=798156,1112951
EC00710=798156,1112951
EC00711=798156,1112951
EC00712=798156,1112951
EC00713=798156,1112951
EC00714=798156,1112951
EC00715=798156,1112951
EC00716=798156,1112951
EC00717=798156,1112951
EC00718=798156,1112951
EC00719=798156,1112951
EC00720=798156,1112951
EC00721=798156,1112951
EC00722=798156,1112951
EC00723=798156,1112951
EC00724=798156,1112951
EC00725=798156,1112951
EC00726=798156,1112951
EC00727=798155,1112950
EC00728=798155,1112950
EC00729=798156,1112951
EC00730=798156,1112951
EC00731=798156,1112951
EC00732=798156,1112951
EC00733=798156,1112951
EC00734=798156,1112951
EC00735=798156,1112951
EC00736=798156,1112951
EC00737=798156,1112951
EC00738=798156,1112951
EC00739=798156,1112951
EC00740=798156,1112951
EC00741=798156,1112951
EC00742=798156,1112951
EC00743=798156,1112951
EC00744=798156,1112951
EC00745=798156,1112951
EC00746=798156,1112951
EC00747=798156,1112951
EC00748=798156,1112951
EC00749=798156,1112951
EC00750=798156,1112951
EC00751=798156,1112951
EC00752=798156,1112951
EC00753=798156,1112951
EC00754=798156,1112951
EC00755=798156,1112951
EC00756=798156,1112951
EC00757=798156,1112951
EC00758=798156,1112951
EC00759=798156,1112951
EC00760=798156,1112951
EC00761=798156,1112951
EC00762=798156,1112951
EC00763=798156,1112951
EC00764=798156,1112951
EC00765=798156,1112951
EC00766=798156,1112951
EC00767=798156,1112951
EC00768=798156,1112951
EC00769=798156,1112951
EC00770=798156,1112951
EC00771=798156,1112951
EC00772=798156,1112951
EC00773=798156,1112951
EC00774=798156,1112951
EC00775=798156,1112951
EC00776=798156,1112951
EC00777=798156,1112951
EC00778=798156,1112951
EC00779=798156,1112951
EC00780=798156,1112951
EC00781=798156,1112951
EC00782=798156,1112951
EC00783=798156,1112951
EC00784=798156,1112951
EC00785=798156,1112951
EC00786=798156,1112951
EC00787=798156,1112951
EC00788=798156,1112951
EC00789=798156,1112951
EC00790=798156,1112951
EC00791=798156,1112951
EC00792=798156,1112951
EC00793=798156,1112951
EC00794=798156,1112951
EC00795=798156,1112951
EC00796=798156,1112951
EC00797=798156,1112951
EC00798=798156,1112951
EC00799=798156,1112951
EC00800=798156,1112951
EC00801=798156,1112951
EC00802=798156,1112951
EC00803=798156,1112951
EC00804=798156,1112951
EC00805=798156,1112951
EC00806=798156,1112951
EC00807=798156,1112951
EC00808=798156,1112951
EC00809=798156,1112951
EC00810=798156,1112951
EC00811=798156,1112951
EC00812=798156,1112951
EC00813=798156,1112951
EC00814=798156,1112951
EC00815=798156,1112951
EC00816=798156,1112951
EC00817=798156,1112951
EC00818=798156,1112951
EC00819=798156,1112951
EC00820=798156,1112951
EC00821=798156,1112951
EC00822=798156,1112951
EC00823=798156,1112951
EC00824=798156,1112951
EC00825=798156,1112951
EC00826=798156,1112951
EC00827=798156,1112951
EC00828=798156,1112951
EC00829=798156,1112951
EC00830=798156,1112951
EC00831=798156,1112951
EC00832=798156,1112951
EC00833=798156,1112951
EC00834=798156,1112951
EC00835=798156,1112951
EC00836=798156,1112951
EC00837=798156,1112951
EC00838=798156,1112951
EC00839=798156,1112951
EC00840=798156,1112951
EC00841=798156,1112951
EC00842=798156,1112951
EC00843=798156,1112951
EC00844=798156,1112951
EC00845=798156,1112951
EC00846=798156,1112951
EC00847=798156,1112951
EC00848=798156,1112951
EC00849=798156,1112951
EC00850=798156,1112951
EC00851=798155,1112950
EC00852=798156,1112951
EC00853=798156,1112951
EC00854=798156,1112951
EC00855=798156,1112951
EC00856=798156,1112951
EC00857=798156,1112951
EC00858=798156,1112951
EC00859=798156,1112951
EC00860=798156,1112951
EC00861=798156,1112951
EC00862=798156,1112951
EC00863=798156,1112951
EC00864=798156,1112951
EC00865=798156,1112951
EC00866=798156,1112951
EC00867=798156,1112951
EC00868=798156,1112951
EC00869=798156,1112951
EC00870=798156,1112951
EC00871=798156,1112951
EC00872=798156,1112951
EC00873=798156,1112951
EC00874=798156,1112951
EC00875=798156,1112951
EC00876=798156,1112951
EC00877=798156,1112951
EC00878=798156,1112951
EC00879=798156,1112951
EC00880=798156,1112951
EC00881=798156,1112951
EC00882=798156,1112951
EC00883=798156,1112951
EC00884=798156,1112951
EC00885=798156,1112951
EC00886=798156,1112951
EC00887=798156,1112951
EC00888=798156,1112951
EC00889=798156,1112951
EC00890=798156,1112951
EC00891=798156,1112951
EC00892=798156,1112951
EC00893=798156,1112951
EC00894=798156,1112951
EC00895=798156,1112951
EC00896=798156,1112951
EC00897=798156,1112951
EC00898=798156,1112951
EC00899=798156,1112951
EC00900=798156,1112951
EC00901=798156,1112951
EC00902=798156,1112951
EC00903=798156,1112951
EC00904=798156,1112951
EC00905=798156,1112951
EC00906=798156,1112951
EC00907=798156,1112951
EC00908=798156,1112951
EC00909=798156,1112951
EC00910=798156,1112951
EC00911=798156,1112951
EC00912=798156,1112951
EC00913=798156,1112951
EC00914=798156,1112951
EC00915=798156,1112951
EC00916=798156,1112951
EC00917=798156,1112951
EC00918=798156,1112951
EC00919=798156,1112951
EC00920=798156,1112951
EC00921=798156,1112951
EC00922=798156,1112951
EC00923=798156,1112951
EC00924=798156,1112951
EC00925=798156,1112951
EC00926=798156,1112951
EC00927=798156,1112951
EC00928=798156,1112951
EC00929=798156,1112951
EC00930=798156,1112951
EC00931=798156,1112951
EC00932=798156,1112951
EC00933=798156,1112951
EC00934=798156,1112951
EC00935=798156,1112951
EC00936=798156,1112951
EC00937=798156,1112951
EC00938=798156,1112951
EC00939=798156,1112951
EC00940=798156,1112951
EC00941=798156,1112951
EC00942=798156,1112951
EC00943=798156,1112951
EC00944=798156,1112951
EC00945=798155,1112951
EC00946=798156,1112951
EC00947=798156,1112951
EC00948=798156,1112951
EC00949=798156,1112951
EC00950=798156,1112951
EC00951=798156,1112951
EC00952=798156,1112951
EC00953=798156,1112951
EC00954=798156,1112951
EC00955=798156,1112951
EC00956=798156,1112951
EC00957=798156,1112951
EC00958=798156,1112951
EC00959=798156,1112951
EC00960=798156,1112951
EC00961=798156,1112951
EC00962=798156,1112951
EC00963=798156,1112951
EC00964=798156,1112951
EC00965=798156,1112951
EC00966=798156,1112951
EC00967=798156,1112951
EC00968=798156,1112951
EC00969=798156,1112951
EC00970=798156,1112951
EC00971=798156,1112951
EC00972=798156,1112951
EC00973=798156,1112951
EC00974=798156,1112951
EC00975=798156,1112951
EC00976=798156,1112951
EC00977=798156,1112951
EC00978=798156,1112951
EC00979=798156,1112951
EC00980=798156,1112951
EC00981=798156,1112951
EC00982=798156,1112951
EC00983=798156,1112951
EC00984=798156,1112951
EC00985=798156,1112951
EC00986=798156,1112951
EC00987=798156,1112951
EC00988=798156,1112951
EC00989=798156,1112951
EC00990=798156,1112951
EC00991=798156,1112951
EC00992=798156,1112951
EC00993=798156,1112951
EC00994=798156,1112951
EC00995=798156,1112951
EC00996=798156,1112951
EC00997=798156,1112951
EC00998=798156,1112951
EC00999=798156,1112951
EC01000=798156,1112951
EC01001=798156,1112951
EC01002=798156,1112951
EC01003=798156,1112951
EC01004=798156,1112951
EC01005=798156,1112951
EC01006=798156,1112951
EC01007=798156,1112951
EC01008=798156,1112951
EC01009=798156,1112951
EC01010=798156,1112951
EC01011=798156,1112951
EC01012=798156,1112951
EC01013=798156,1112951
EC01014=798156,1112951
EC01015=798156,1112951
EC01016=798156,1112951
EC01017=798156,1112951
EC01018=798156,1112951
EC01019=798156,1112951
EC01020=798156,1112951
EC01021=798156,1112951
EC01022=798156,1112951
EC01023=798156,1112951
EC01024=798156,1112951
EC01025=798156,1112951
EC01026=798156,1112951
EC01027=798156,1112951
EC01028=798156,1112951
EC01029=798156,1112951
EC01030=798156,1112951
EC01031=798155,1112950
EC01032=798155,1112950
EC01033=798156,1112951
EC01034=798156,1112951
EC01035=798156,1112951
EC01036=798156,1112951
EC01037=798156,1112951
EC01038=798156,1112951
EC01039=798155,1112951
EC01040=798155,1112951
EC01041=798156,1112951
EC01042=798156,1112951
EC01043=798156,1112951
EC01044=798156,1112951
EC01045=798156,1112951
EC01046=798156,1112951
EC01047=798156,1112951
EC01048=798156,1112951
EC01049=798155,1112950
EC01050=798156,1112951
EC01051=798156,1112951
EC01052=798156,1112951
EC01053=798156,1112951
EC01054=798156,1112951
EC01055=798156,1112951
EC01056=798156,1112951
EC01057=798156,1112951
EC01058=798156,1112951
EC01059=798156,1112951
EC01060=798156,1112951
EC01061=798156,1112951
EC01062=798156,1112951
EC01063=798156,1112951
EC01064=798156,1112951
EC01065=798156,1112951
EC01066=798155,1112950
EC01067=798156,1112951
EC01068=798156,1112951
EC01069=798156,1112951
EC01070=798156,1112951
EC01071=798156,1112951
EC01072=798156,1112951
EC01073=798156,1112951
EC01074=798156,1112951
EC01075=798156,1112951
EC01076=798156,1112951
EC01077=798155,1112950
EC01078=798156,1112951
EC01079=798156,1112951
EC01080=798156,1112951
EC01081=798156,1112951
EC01082=798156,1112951
EC01083=798156,1112951
EC01084=798156,1112951
EC01085=798156,1112951
EC01086=798156,1112951
EC01087=798156,1112951
EC01088=798156,1112951
EC01089=798156,1112951
EC01090=798156,1112951
EC01091=798156,1112951
EC01092=798156,1112951
EC01093=798156,1112951
EC01094=798156,1112951
EC01095=798156,1112951
EC01096=798156,1112951
EC01097=798156,1112951
EC01098=798156,1112951
EC01099=798156,1112951
EC01100=798156,1112951
EC01101=798156,1112951
EC01102=798156,1112951
EC01103=798156,1112951
EC01104=798156,1112951
EC01105=798156,1112951
EC01106=798156,1112951
EC01107=798156,1112951
EC01108=798156,1112951
EC01109=798156,1112951
EC01110=798156,1112951
EC01111=798156,1112951
EC01112=798155,1112950
EC01113=798156,1112951
EC01114=798156,1112951
EC01115=798156,1112951
EC01116=798156,1112951
EC01117=798156,1112951
EC01118=798156,1112951
EC01119=798156,1112951
EC01120=798156,1112951
EC01121=798156,1112951
EC01122=798156,1112951
EC01123=798156,1112951
EC01124=798156,1112951
EC01125=798156,1112951
EC01126=798156,1112951
EC01127=798156,1112951
EC01128=798156,1112951
EC01129=798156,1112951
EC01130=798156,1112951
EC01131=798156,1112951
EC01132=798156,1112951
EC01133=798156,1112951
EC01134=798156,1112951
EC01135=798156,1112951
EC01136=798156,1112951
EC01137=798156,1112951
EC01138=798156,1112951
EC01139=798156,1112951
EC01140=798156,1112951
EC01141=798156,1112951
EC01142=798156,1112951
EC01143=798156,1112951
EC01144=798156,1112951
EC01145=798156,1112951
EC01146=798156,1112951
EC01147=798156,1112951
EC01148=798156,1112951
EC01149=798156,1112951
EC01150=798156,1112951
EC01151=798156,1112951
EC01152=798156,1112951
EC01153=798156,1112951
EC01154=798156,1112951
EC01155=798156,1112951
EC01156=798156,1112951
EC01157=798156,1112951
EC01158=798156,1112951
EC01159=798156,1112951
EC01160=798156,1112951
EC01161=798156,1112951
EC01162=798156,1112951
EC01163=798156,1112951
EC01164=798156,1112951
EC01165=798156,1112951
EC01166=798156,1112951
EC01167=798156,1112951
EC01168=798156,1112951
EC01169=798156,1112951
EC01170=798156,1112951
EC01171=798156,1112951
EC01172=798156,1112951
EC01173=798156,1112951
EC01174=798156,1112951
EC01175=798156,1112951
EC01176=798156,1112951
EC01177=798155,1112951
EC01178=798156,1112951
EC01179=798156,1112951
EC01180=798156,1112951
EC01181=798156,1112951
EC01182=798156,1112951
EC01183=798156,1112951
EC01184=798156,1112951
EC01185=798156,1112951
EC01186=798156,1112951
EC01187=798156,1112951
EC01188=798156,1112951
EC01189=798156,1112951
EC01190=798156,1112951
EC01191=798156,1112951
EC01192=798156,1112951
EC01193=798156,1112951
EC01194=798156,1112951
EC01195=798156,1112951
EC01196=798156,1112951
EC01197=798156,1112951
EC01198=798156,1112951
EC01199=798156,1112951
EC01200=798156,1112951
EC01201=798156,1112951
EC01202=798156,1112951
EC01203=798156,1112951
EC01204=798156,1112951
EC01205=798156,1112951
EC01206=798156,1112951
EC01207=798156,1112951
EC01208=798156,1112951
EC01209=798156,1112951
EC01210=798156,1112951
EC01211=798156,1112951
EC01212=798156,1112951
EC01213=798156,1112951
EC01214=798156,1112951
EC01215=798156,1112951
EC01216=798156,1112951
EC01217=798156,1112951
EC01218=798156,1112951
EC01219=798156,1112951
EC01220=798156,1112951
EC01221=798156,1112951
EC01222=798156,1112951
EC01223=798156,1112951
EC01224=798156,1112951
EC01225=798156,1112951
EC01226=798156,1112951
EC01227=798156,1112951
EC01228=798156,1112951
EC01229=798156,1112951
EC01230=798156,1112951
EC01231=798156,1112951
EC01232=798156,1112951
EC01233=798156,1112951
EC01234=798156,1112951
EC01235=798156,1112951
EC01236=798156,1112951
EC01237=798156,1112951
EC01238=798156,1112951
EC01239=798156,1112951
EC01240=798156,1112951
EC01241=798156,1112951
EC01242=798156,1112951
EC01243=798156,1112951
EC01244=798156,1112951
EC01245=798156,1112951
EC01246=798156,1112951
EC01247=798156,1112951
EC01248=798156,1112951
EC01249=798156,1112951
EC01250=798156,1112951
EC01251=798156,1112951
EC01252=798156,1112951
EC01253=798156,1112951
EC01254=798156,1112951
EC01255=798156,1112951
EC01256=798156,1112951
EC01257=798156,1112951
EC01258=798156,1112951
EC01259=798156,1112951
EC01260=798156,1112951
EC01261=798156,1112951
EC01262=798156,1112951
EC01263=798156,1112951
EC01264=798156,1112951
EC01265=798156,1112951
EC01266=798156,1112951
EC01267=798156,1112951
EC01268=798156,1112951
EC01269=798156,1112951
EC01270=798156,1112951
EC01271=798156,1112951
EC01272=798156,1112951
EC01273=798156,1112951
EC01274=798156,1112951
EC01275=798156,1112951
EC01276=798156,1112951
EC01277=798156,1112951
EC01278=798156,1112951
EC01279=798156,1112951
EC01280=798156,1112951
EC01281=798156,1112951
EC01282=798156,1112951
EC01283=798156,1112951
EC01284=798156,1112951
EC01285=798156,1112951
EC01286=798156,1112951
EC01287=798156,1112951
EC01288=798156,1112951
EC01289=798156,1112951
EC01290=798156,1112951
EC01291=798156,1112951
EC01292=798156,1112951
EC01293=798156,1112951
EC01294=798156,1112951
EC01295=798156,1112951
EC01296=798156,1112951
EC01297=798156,1112951
EC01298=798156,1112951
EC01299=798156,1112951
EC01300=798156,1112951
EC01301=798156,1112951
EC01302=798156,1112951
EC01303=798156,1112951
EC01304=798156,1112951
EC01305=798155,1112950
EC01306=798156,1112951
EC01307=798156,1112951
EC01308=798156,1112951
EC01309=798156,1112951
EC01310=798156,1112951
EC01311=798156,1112951
EC01312=798156,1112951
EC01313=798156,1112951
EC01314=798156,1112951
EC01315=798156,1112951
EC01316=798156,1112951
EC01317=798156,1112951
EC01318=798156,1112951
EC01319=798156,1112951
EC01320=798156,1112951
EC01321=798156,1112951
EC01322=798156,1112951
EC01323=798156,1112951
EC01324=798156,1112951
EC01325=798156,1112951
EC01326=798156,1112951
EC01327=798156,1112951
EC01328=798156,1112951
EC01329=798156,1112951
EC01330=798156,1112951
EC01331=798156,1112951
EC01332=798156,1112951
EC01333=798156,1112951
EC01334=798156,1112951
EC01335=798156,1112951
EC01336=798156,1112951
EC01337=798156,1112951
EC01338=798156,1112951
EC01339=798156,1112951
EC01340=798156,1112951
EC01341=798156,1112951
EC01342=798156,1112951
EC01343=798156,1112951
EC01344=798156,1112951
EC01345=798156,1112951
EC01346=798156,1112951
EC01347=798156,1112951
EC01348=798156,1112951
EC01349=798156,1112951
EC01350=798156,1112951
EC01351=798156,1112951
EC01352=798156,1112951
EC01353=798156,1112951
EC01354=798156,1112951
EC01355=798156,1112951
EC01356=798156,1112951
EC01357=798156,1112951
EC01358=798156,1112951
EC01359=798156,1112951
EC01360=798156,1112951
EC01361=798156,1112951
EC01362=798156,1112951
EC01363=798156,1112951
EC01364=798156,1112951
EC01365=798156,1112951
EC01366=798156,1112951
EC01367=798156,1112951
EC01368=798156,1112951
EC01369=798156,1112951
EC01370=798156,1112951
EC01371=798156,1112951
EC01372=798156,1112951
EC01373=798156,1112951
EC01374=798156,1112951
EC01375=798156,1112951
EC01376=798156,1112951
EC01377=798156,1112951
EC01378=798156,1112951
EC01379=798156,1112951
EC01380=798156,1112951
EC01381=798156,1112951
EC01382=798156,1112951
EC01383=798156,1112951
EC01384=798156,1112951
EC01385=798156,1112951
EC01386=798156,1112951
EC01387=798156,1112951
EC01388=798156,1112951
EC01389=798156,1112951
EC01390=798156,1112951
EC01391=798156,1112951
EC01392=798156,1112951
EC01393=798156,1112951
EC01394=798156,1112951
EC01395=798156,1112951
EC01396=798156,1112951
EC01397=798156,1112951
EC01398=798156,1112951
EC01399=798156,1112951
EC01400=798156,1112951
EC01401=798156,1112951
EC01402=798156,1112951
EC01403=798156,1112951
EC01404=798156,1112951
EC01405=798156,1112951
EC01406=798156,1112951
EC01407=798156,1112951
EC01408=798156,1112951
EC01409=798156,1112951
EC01410=798156,1112951
EC01411=798156,1112951
EC01412=798156,1112951
EC01413=798156,1112951
EC01414=798156,1112951
EC01415=798156,1112951
EC01416=798156,1112951
EC01417=798156,1112951
EC01418=798156,1112951
EC01419=798156,1112951
EC01420=798156,1112951
EC01421=798156,1112951
EC01422=798156,1112951
EC01423=798156,1112951
EC01424=798156,1112951
EC01425=798156,1112951
EC01426=798156,1112951
EC01427=798155,1112951
EC01428=798155,1112951
EC01429=798156,1112951
EC01430=798156,1112951
EC01431=798156,1112951
EC01432=798156,1112951
EC01433=798156,1112951
EC01434=798156,1112951
EC01435=798156,1112951
EC01436=798156,1112951
EC01437=798155,1112950
EC01438=798155,1112950
EC01439=798155,1112950
EC01440=798155,1112950
EC01441=798155,1112950
EC01442=798156,1112951
EC01443=798156,1112951
EC01444=798156,1112951
EC01445=798156,1112951
EC01446=798156,1112951
EC01447=798156,1112951
EC01448=798156,1112951
EC01449=798156,1112951
EC01450=798156,1112951
EC01451=798156,1112951
EC01452=798156,1112951
EC01453=798156,1112951
EC01454=798156,1112951
EC01455=798156,1112951
EC01456=798156,1112951
EC01457=798156,1112951
EC01458=798156,1112951
EC01459=798156,1112951
EC01460=798156,1112951
EC01461=798156,1112951
EC01462=798156,1112951
EC01463=798156,1112951
EC01464=798156,1112951
EC01465=798156,1112951
EC01466=798156,1112951
EC01467=798156,1112951
EC01468=798156,1112951
EC01469=798156,1112951
EC01470=798156,1112951
EC01471=798156,1112951
EC01472=798156,1112951
EC01473=798156,1112951
EC01474=798156,1112951
EC01475=798156,1112951
EC01476=798156,1112951
EC01477=798156,1112951
EC01478=798156,1112951
EC01479=798156,1112951
EC01480=798156,1112951
EC01481=798156,1112951
EC01482=798156,1112951
EC01483=798156,1112951
EC01484=798156,1112951
EC01485=798156,1112951
EC01486=798156,1112951
EC01487=798156,1112951
EC01488=798156,1112951
EC01489=798156,1112951
EC01490=798156,1112951
EC01491=798156,1112951
EC01492=798156,1112951
EC01493=798156,1112951
EC01494=798156,1112951
EC01495=798156,1112951
EC01496=798156,1112951
EC01497=798156,1112951
EC01498=798156,1112951
EC01499=798156,1112951
EC01500=798156,1112951
EC01501=798156,1112951
EC01502=798156,1112951
EC01503=798156,1112951
EC01504=798156,1112951
EC01505=798156,1112951
EC01506=798156,1112951
EC01507=798156,1112951
EC01508=798156,1112951
EC01509=798156,1112951
EC01510=798156,1112951
EC01511=798156,1112951
EC01512=798155,1112950
EC01513=798155,1112950
EC01514=798155,1112950
EC01515=798155,1112950
EC01516=798155,1112950
EC01517=798155,1112950
EC01518=798155,1112950
EC01519=798155,1112950
EC01520=798155,1112950
EC01521=798155,1112950
EC01522=798155,1112950
EC01523=798155,1112950
EC01524=798155,1112950
EC01525=798156,1112951
EC01526=798156,1112951
EC01527=798156,1112951
EC01528=798156,1112951
EC01529=798156,1112951
EC01530=798156,1112951
EC01531=798155,1112950
EC01532=798155,1112950
EC01533=798155,1112950
EC01534=798155,1112950
EC01535=798155,1112950
EC01536=798155,1112950
EC01537=798155,1112950
EC01538=798155,1112950
EC01539=798154,1112949
EC01540=798154,1112949
EC01541=798154,1112949
EC01542=798154,1112949
EC01543=798156,1112951
EC01544=798156,1112951
EC01545=798156,1112951
EC01546=798156,1112951
EC01547=798156,1112951
EC01548=798156,1112951
EC01549=798156,1112951
EC01550=798156,1112951
EC01551=798156,1112951
EC01552=798156,1112951
EC01553=798156,1112951
EC01554=798156,1112951
EC01555=798156,1112951
EC01556=798156,1112951
EC01557=798156,1112951
EC01558=798156,1112951
EC01559=798156,1112951
EC01560=798156,1112951
EC01561=798156,1112951
EC01562=798156,1112951
EC01563=798156,1112951
EC01564=798156,1112951
EC01565=798156,1112951
EC01566=798156,1112951
EC01567=798156,1112951
EC01568=798156,1112951
EC01569=798156,1112951
EC01570=798156,1112951
EC01571=798156,1112951
EC01572=798156,1112951
EC01573=798156,1112951
EC01574=798156,1112951
EC01575=798156,1112951
EC01576=798156,1112951
EC01577=798156,1112951
EC01578=798156,1112951
EC01579=798156,1112951
EC01580=798156,1112951
EC01581=798156,1112951
EC01582=798156,1112951
EC01583=798156,1112951
EC01584=798156,1112951
EC01585=798156,1112951
EC01586=798156,1112951
EC01587=798156,1112949
EC01588=798156,1112951
EC01589=798156,1112951
EC01590=798156,1112951
EC01591=798156,1112951
EC01592=798156,1112951
EC01593=798156,1112951
EC01594=798156,1112951
EC01595=798156,1112951
EC01596=798156,1112951
EC01597=798156,1112951
EC01598=798156,1112951
EC01599=798156,1112951
EC01600=798156,1112951
EC01601=798156,1112951
EC01602=798156,1112951
EC01603=798156,1112951
EC01604=798156,1112951
EC01605=798156,1112951
EC01606=798156,1112951
EC01607=798156,1112951
EC01608=798156,1112951
EC01609=798156,1112951
EC01610=798156,1112951
EC01611=798156,1112951
EC01612=798156,1112951
EC01613=798156,1112951
EC01614=798156,1112951
EC01615=798156,1112951
EC01616=798156,1112951
EC01617=798156,1112951
EC01618=798156,1112951
EC01619=798156,1112951
EC01620=798156,1112951
EC01621=798156,1112951
EC01622=798156,1112951
EC01623=798156,1112951
EC01624=798156,1112951
EC01625=798156,1112951
EC01626=798156,1112951
EC01627=798156,1112951
EC01628=798156,1112951
EC01629=798156,1112951
EC01630=798156,1112951
EC01631=798156,1112951
EC01632=798156,1112951
EC01633=798156,1112951
EC01634=798156,1112951
EC01635=798156,1112951
EC01636=798156,1112951
EC01637=798156,1112951
EC01638=798156,1112951
EC01639=798156,1112951
EC01640=798156,1112951
EC01641=798156,1112951
EC01642=798156,1112951
EC01643=798156,1112951
EC01644=798156,1112951
EC01645=798156,1112951
EC01646=798156,1112951
EC01647=798156,1112951
EC01648=798156,1112951
EC01649=798156,1112951
EC01650=798156,1112951
EC01651=798156,1112951
EC01652=798155,1112950
EC01653=798155,1112950
EC01654=798155,1112950
EC01655=798155,1112950
EC01656=798155,1112950
EC01657=798155,1112950
EC01658=798155,1112950
EC01659=798156,1112951
EC01660=798156,1112951
EC01661=798156,1112951
EC01662=798156,1112951
EC01663=798156,1112951
EC01664=798156,1112951
EC01665=798156,1112951
EC01666=798156,1112951
EC01667=798156,1112951
EC01668=798156,1112951
EC01669=798156,1112951
EC01670=798156,1112951
EC01671=798156,1112951
EC01672=798156,1112951
EC01673=798156,1112951
EC01674=798156,1112951
EC01675=798156,1112951
EC01676=798156,1112951
EC01677=798156,1112951
EC01678=798156,1112951
EC01679=798156,1112951
EC01680=798156,1112951
EC01681=798156,1112951
EC01682=798156,1112951
EC01683=798156,1112951
EC01684=798156,1112951
EC01685=798156,1112951
EC01686=798156,1112951
EC01687=798156,1112951
EC01688=798156,1112951
EC01689=798156,1112951
EC01690=798156,1112951
EC01691=798156,1112951
EC01692=798156,1112951
EC01693=798156,1112951
EC01694=798156,1112951
EC01695=798156,1112951
EC01696=798156,1112951
EC01697=798156,1112951
EC01698=798156,1112951
EC01699=798156,1112951
EC01700=798156,1112951
EC01701=798156,1112951
EC01702=798156,1112951
EC01703=798156,1112951
EC01704=798156,1112951
EC01705=798156,1112951
EC01706=798156,1112951
EC01707=798156,1112951
EC01708=798156,1112951
EC01709=798156,1112951
EC01710=798156,1112951
EC01711=798156,1112951
EC01712=798156,1112951
EC01713=798156,1112951
EC01714=798156,1112951
EC01715=798156,1112951
EC01716=798156,1112951
EC01717=798156,1112951
EC01718=798156,1112951
EC01719=798156,1112951
EC01720=798156,1112951
EC01721=798156,1112951
EC01722=798156,1112951
EC01723=798156,1112951
EC01724=798156,1112951
EC01725=798156,1112951
EC01726=798155,1112949
EC01727=798156,1112951
EC01728=798156,1112951
EC01729=798156,1112951
EC01730=798156,1112951
EC01731=798156,1112951
EC01732=798156,1112951
EC01733=798156,1112951
EC01734=798156,1112951
EC01735=798156,1112951
EC01736=798156,1112951
EC01737=798156,1112951
EC01738=798156,1112951
EC01739=798156,1112951
EC01740=798156,1112951
EC01741=798156,1112951
EC01742=798156,1112951
EC01743=798156,1112951
EC01744=798156,1112951
///POSTYPE BASE
///RECTAN
///RCONF 0,0,0,0,0,0,0,0,0,0,0,0,0,0,0,0,0,0,0,0,0,0,0,0
P00006=0.000,0.000,0.000,0.0000,0.0000,0.0000
P00021=3.198,-0.012,-3.236,0.0000,0.0000,0.0000
P00022=-0.007,0.008,-4.232,0.0000,0.0000,0.0000
P00023=0.143,-0.036,0.682,0.0000,0.0000,0.0000
P00024=0.145,-0.552,1.326,0.0000,0.0000,0.0000
P00025=-2.003,0.006,0.728,0.0000,0.0000,0.0000
P00026=0.562,-0.002,-0.337,0.0000,0.0000,0.0000
P00027=-0.746,0.015,-9.096,0.0000,0.0000,0.0000
P00028=-2.237,-0.018,-7.702,0.0000,0.0000,0.0000
P00029=-2.156,-0.086,-4.681,0.0000,0.0000,0.0000
P00030=5.926,-4.294,-1.390,0.0000,0.0000,0.0000
P00031=1.853,-0.001,-1.549,0.0000,0.0000,0.0000
P00032=1.957,0.503,-7.217,0.0000,0.0000,0.0000
///RCONF 0,0,0,0,1,0,0,0,0,0,0,0,0,0,0,0,0,0,0,0,0,0,0,0
P00033=-0.123,0.612,-5.012,0.0000,0.0000,0.0000
///RCONF 0,0,0,0,0,0,0,0,0,0,0,0,0,0,0,0,0,0,0,0,0,0,0,0
P00034=-0.304,0.773,-2.693,0.0000,0.0000,0.0000
P00035=2.817,0.591,-1.622,0.0000,0.0000,0.0000
P00040=-0.030,9.648,2.467,0.0000,0.0000,0.0000
P00041=0.192,3.924,0.305,0.0000,0.0000,0.0000
P00042=-0.217,1.941,0.413,0.0000,0.0000,0.0000
P00043=-0.044,-1.937,1.197,0.0000,0.0000,0.0000
P00044=0.687,-2.322,1.156,0.0000,0.0000,0.0000
P00045=-0.068,-0.810,1.603,0.0000,0.0000,0.0000
P00046=0.799,0.043,1.292,0.0000,0.0000,0.0000
///RCONF 0,1,0,0,0,0,0,0,0,0,0,0,0,0,0,0,0,0,0,0,0,0,0,0
P00047=-0.011,1.737,-0.646,0.0000,0.0000,0.0000
///RCONF 0,0,0,0,0,0,0,0,0,0,0,0,0,0,0,0,0,0,0,0,0,0,0,0
P00048=2.411,0.025,-0.606,0.0000,0.0000,0.0000
P00049=3.413,-3.572,-1.618,0.0000,0.0000,0.0000
P00050=4.296,-4.501,-0.826,0.0000,0.0000,0.0000
P00051=0.367,3.892,0.009,0.0000,0.0000,0.0000
P00052=0.088,2.832,-0.342,0.0000,0.0000,0.0000
P00053=0.134,6.594,0.107,0.0000,0.0000,0.0000
P00054=-0.103,6.509,-0.702,0.0000,0.0000,0.0000
P00055=-0.342,8.912,1.324,0.0000,0.0000,0.0000
P00061=1.575,-3.405,-0.752,0.0000,0.0000,0.0000
P00062=-0.135,-0.848,-1.706,0.0000,0.0000,0.0000
P00063=0.036,-0.654,-3.005,0.0000,0.0000,0.0000
P00071=2.716,0.070,1.352,0.0000,0.0000,0.0000
P00072=1.041,-0.003,-0.797,0.0000,0.0000,0.0000
P00073=-0.961,5.319,-6.157,0.0000,0.0000,0.0000
P00074=1.123,1.944,-5.914,0.0000,0.0000,0.0000
P00080=-3.893,-3.240,-0.208,0.0000,0.0000,0.0000
P00081=19.486,11.347,1.262,0.0000,0.0000,0.0000
P00088=-2.376,0.094,2.453,0.0000,0.0000,0.0000
P00089=5.697,-3.100,-1.263,0.0000,0.0000,0.0000
P00095=-3.945,4.918,-0.177,0.0000,0.0000,0.0000
P00096=-0.633,5.398,-3.809,0.0000,0.0000,0.0000
P00097=0.069,0.776,0.128,0.0000,0.0000,0.0000
P00098=0.276,2.477,1.230,0.0000,0.0000,0.0000
//INST
///DATE 2025/03/11 14:50
///ATTR SC,RW
///GROUP1 RB1,BS1
///GROUP2 ST1
NOP
COMM 'X2_8B-21B(90,180)
COMM '
COMM MOVJ C00000 BC00000 VJ=100.00  +MOVJ EC00000 VJ=100.00
COMM 'Path S4722
COMM SFTOF3D
COMM MOVJ C00001 BC00001 VJ=100.00  +MOVJ EC00001 VJ=100.00
COMM MOVL C00002 BC00002 V=666.7  +MOVJ EC00002 VJ=100.00
COMM SMOVL C00003 BC00003 V=166.7  +MOVJ EC00003
COMM SREFP 3 C00004 BC00004  +REFP EC00004
COMM CALL JOB:SEARCH-R1-S13D
COMM SET P095 P006
COMM SFTON3D P095
COMM SMOVL C00005 BC00005 V=166.7  +MOVJ EC00005
COMM SREFP 3 C00006 BC00006  +REFP EC00006
COMM CALL JOB:SEARCH-R1-S13D
COMM SET P095 P006
COMM SFTON3D P095
COMM SMOVL C00007 BC00007 V=166.7  +MOVJ EC00007
COMM MOVL C00008 BC00008 V=1000.0  +MOVJ EC00008 VJ=100.00
COMM 'EndPath S4722
COMM 'Path S4723
COMM SFTOF3D
COMM MOVJ C00009 BC00009 VJ=100.00  +MOVJ EC00009 VJ=100.00
COMM MOVL C00010 BC00010 V=666.7  +MOVJ EC00010 VJ=100.00
COMM SMOVL C00011 BC00011 V=166.7  +MOVJ EC00011
COMM SREFP 3 C00012 BC00012  +REFP EC00012
COMM CALL JOB:SEARCH-R1-S13D
COMM SET P096 P006
COMM SFTON3D P096
COMM SMOVL C00013 BC00013 V=166.7  +MOVJ EC00013
COMM SREFP 3 C00014 BC00014  +REFP EC00014
COMM CALL JOB:SEARCH-R1-S13D
COMM SET P096 P006
COMM SFTON3D P096
COMM SMOVL C00015 BC00015 V=166.7  +MOVJ EC00015
COMM MOVL C00016 BC00016 V=1000.0  +MOVJ EC00016 VJ=100.00
COMM 'EndPath S4723
COMM '
COMM '
COMM 'Path S4093
COMM SFTOF3D
COMM MOVJ C00017 BC00017 VJ=100.00  +MOVJ EC00017 VJ=100.00
COMM MOVL C00018 BC00018 V=666.7  +MOVJ EC00018 VJ=100.00
COMM SMOVL C00019 BC00019 V=166.7  +MOVJ EC00019
COMM SREFP 3 C00020 BC00020  +REFP EC00020
COMM CALL JOB:SEARCH-R1-S13D
COMM SET P021 P006
COMM SFTON3D P021
COMM SMOVL C00021 BC00021 V=166.7  +MOVJ EC00021
COMM SREFP 3 C00022 BC00022  +REFP EC00022
COMM CALL JOB:SEARCH-R1-S13D
COMM SET P021 P006
COMM SFTON3D P021
COMM SMOVL C00023 BC00023 V=166.7  +MOVJ EC00023
COMM MOVL C00024 BC00024 V=1000.0  +MOVJ EC00024 VJ=100.00
COMM 'EndPath S4093
COMM 'Path S4094
COMM SFTOF3D
COMM MOVJ C00025 BC00025 VJ=100.00  +MOVJ EC00025 VJ=100.00
COMM MOVL C00026 BC00026 V=666.7  +MOVJ EC00026 VJ=100.00
COMM SMOVL C00027 BC00027 V=166.7  +MOVJ EC00027
COMM SREFP 3 C00028 BC00028  +REFP EC00028
COMM CALL JOB:SEARCH-R1-S13D
COMM SET P022 P006
COMM SFTON3D P022
COMM SMOVL C00029 BC00029 V=166.7  +MOVJ EC00029
COMM SREFP 3 C00030 BC00030  +REFP EC00030
COMM CALL JOB:SEARCH-R1-S13D
COMM SET P022 P006
COMM SFTON3D P022
COMM SMOVL C00031 BC00031 V=166.7  +MOVJ EC00031
COMM MOVL C00032 BC00032 V=1000.0  +MOVJ EC00032 VJ=100.00
COMM 'EndPath S4094
COMM MOVJ C00033 BC00033 VJ=100.00  +MOVJ EC00033 VJ=100.00
COMM 'Path S4205
COMM SFTOF3D
COMM MOVJ C00034 BC00034 VJ=100.00  +MOVJ EC00034 VJ=100.00
COMM MOVL C00035 BC00035 V=666.7  +MOVJ EC00035 VJ=100.00
COMM SMOVL C00036 BC00036 V=166.7  +MOVJ EC00036
COMM SREFP 3 C00037 BC00037  +REFP EC00037
COMM CALL JOB:SEARCH-R1-S13D
COMM SET P050 P006
COMM SFTON3D P050
COMM SMOVL C00038 BC00038 V=166.7  +MOVJ EC00038
COMM SREFP 3 C00039 BC00039  +REFP EC00039
COMM CALL JOB:SEARCH-R1-S13D
COMM SET P050 P006
COMM SFTON3D P050
COMM SMOVL C00040 BC00040 V=166.7  +MOVJ EC00040
COMM SMOVL C00041 BC00041 V=250.0  +MOVJ EC00041
COMM SMOVL C00042 BC00042 V=166.7  +MOVJ EC00042
COMM SREFP 3 C00043 BC00043  +REFP EC00043
COMM CALL JOB:SEARCH-R1-S13D
COMM SET P050 P006
COMM SFTON3D P050
COMM SMOVL C00044 BC00044 V=250.0  +MOVJ EC00044
COMM 'EndPath S4205
COMM 'Path S4206
COMM SFTOF3D
COMM MOVL C00045 BC00045 V=1000.0  +MOVJ EC00045 VJ=100.00
COMM SMOVL C00046 BC00046 V=166.7  +MOVJ EC00046
COMM SREFP 3 C00047 BC00047  +REFP EC00047
COMM CALL JOB:SEARCH-R1-S13D
COMM SET P051 P006
COMM SFTON3D P051
COMM SMOVL C00048 BC00048 V=166.7  +MOVJ EC00048
COMM SREFP 3 C00049 BC00049  +REFP EC00049
COMM CALL JOB:SEARCH-R1-S13D
COMM SET P051 P006
COMM SFTON3D P051
COMM SMOVL C00050 BC00050 V=166.7  +MOVJ EC00050
COMM SMOVL C00051 BC00051 V=250.0  +MOVJ EC00051
COMM SREFP 3 C00052 BC00052  +REFP EC00052
COMM CALL JOB:SEARCH-R1-S13D
COMM SET P051 P006
COMM SFTON3D P051
COMM SMOVL C00053 BC00053 V=250.0  +MOVJ EC00053
COMM MOVL C00054 BC00054 V=1000.0  +MOVJ EC00054 VJ=100.00
COMM 'EndPath S4206
COMM MOVJ C00055 BC00055 VJ=100.00  +MOVJ EC00055 VJ=100.00
COMM 'Path S4207
COMM SFTOF3D
COMM MOVJ C00056 BC00056 VJ=100.00  +MOVJ EC00056 VJ=100.00
COMM MOVL C00057 BC00057 V=666.7  +MOVJ EC00057 VJ=100.00
COMM SMOVL C00058 BC00058 V=166.7  +MOVJ EC00058
COMM SREFP 3 C00059 BC00059  +REFP EC00059
COMM CALL JOB:SEARCH-R1-S13D
COMM SET P054 P006
COMM SFTON3D P054
COMM SMOVL C00060 BC00060 V=250.0  +MOVJ EC00060
COMM SMOVL C00061 BC00061 V=233.3  +MOVJ EC00061
COMM SMOVL C00062 BC00062 V=166.7  +MOVJ EC00062
COMM SREFP 3 C00063 BC00063  +REFP EC00063
COMM CALL JOB:SEARCH-R1-S13D
COMM SET P054 P006
COMM SFTON3D P054
COMM SMOVL C00064 BC00064 V=166.7  +MOVJ EC00064
COMM SMOVL C00065 BC00065 V=416.7  +MOVJ EC00065
COMM SMOVL C00066 BC00066 V=250.0  +MOVJ EC00066
COMM SREFP 3 C00067 BC00067  +REFP EC00067
COMM CALL JOB:SEARCH-R1-S13D
COMM SET P054 P006
COMM SFTON3D P054
COMM SMOVL C00068 BC00068 V=250.0  +MOVJ EC00068
COMM MOVL C00069 BC00069 V=1000.0  +MOVJ EC00069 VJ=100.00
COMM 'EndPath S4207
COMM 'Path S4095
COMM SFTOF3D
COMM MOVJ C00070 BC00070 VJ=100.00  +MOVJ EC00070 VJ=100.00
COMM MOVJ C00071 BC00071 VJ=100.00  +MOVJ EC00071 VJ=100.00
COMM SMOVL C00072 BC00072 V=200.0  +MOVJ EC00072
COMM SREFP 3 C00073 BC00073  +REFP EC00073
COMM CALL JOB:SEARCH-R1-S13D
COMM SET P089 P006
COMM SFTON3D P089
COMM SMOVL C00074 BC00074 V=166.7  +MOVJ EC00074
COMM SMOVL C00075 BC00075 V=166.7  +MOVJ EC00075
COMM SREFP 3 C00076 BC00076  +REFP EC00076
COMM CALL JOB:SEARCH-R1-S13D
COMM SET P089 P006
COMM SFTON3D P089
COMM SMOVL C00077 BC00077 V=166.7  +MOVJ EC00077
COMM SMOVL C00078 BC00078 V=166.7  +MOVJ EC00078
COMM SREFP 3 C00079 BC00079  +REFP EC00079
COMM CALL JOB:SEARCH-R1-S13D
COMM SET P089 P006
COMM SFTON3D P089
COMM SMOVL C00080 BC00080 V=166.7  +MOVJ EC00080
COMM SMOVL C00081 BC00081 V=1000.0  +MOVJ EC00081
COMM SFTOF3D
COMM MOVJ C00082 BC00082 VJ=100.00  +MOVJ EC00082 VJ=100.00
COMM MOVL C00083 BC00083 V=666.7  +MOVJ EC00083 VJ=100.00
COMM SMOVL C00084 BC00084 V=166.7  +MOVJ EC00084
COMM SREFP 3 C00085 BC00085  +REFP EC00085
COMM CALL JOB:SEARCH-R1-S13D
COMM SET P034 P006
COMM SFTON3D P034
COMM SMOVL C00086 BC00086 V=250.0  +MOVJ EC00086
COMM SMOVL C00087 BC00087 V=233.3  +MOVJ EC00087
COMM SMOVL C00088 BC00088 V=166.7  +MOVJ EC00088
COMM SREFP 3 C00089 BC00089  +REFP EC00089
COMM CALL JOB:SEARCH-R1-S13D
COMM SET P034 P006
COMM SFTON3D P034
COMM SMOVL C00090 BC00090 V=166.7  +MOVJ EC00090
COMM SMOVL C00091 BC00091 V=166.7  +MOVJ EC00091
COMM SREFP 3 C00092 BC00092  +REFP EC00092
COMM CALL JOB:SEARCH-R1-S13D
COMM SET P034 P006
COMM SFTON3D P034
COMM SMOVL C00093 BC00093 V=166.7  +MOVJ EC00093
COMM MOVJ C00094 BC00094 VJ=50.00  +MOVJ EC00094 VJ=30.00
COMM 'EndPath S4095
COMM 'Path S4096
COMM SFTOF3D
COMM MOVJ C00095 BC00095 VJ=50.00  +MOVJ EC00095 VJ=30.00
COMM MOVJ C00096 BC00096 VJ=50.00  +MOVJ EC00096 VJ=30.00
COMM MOVJ C00097 BC00097 VJ=50.00  +MOVJ EC00097 VJ=30.00
COMM SMOVL C00098 BC00098 V=166.7  +MOVJ EC00098
COMM SREFP 3 C00099 BC00099  +REFP EC00099
COMM CALL JOB:SEARCH-R1-S13D
COMM SET P061 P006
COMM SFTON3D P061
COMM SMOVL C00100 BC00100 V=166.7  +MOVJ EC00100
COMM SREFP 3 C00101 BC00101  +REFP EC00101
COMM CALL JOB:SEARCH-R1-S13D
COMM SET P061 P006
COMM SFTON3D P061
COMM SMOVL C00102 BC00102 V=166.7  +MOVJ EC00102
COMM SFTOF3D
COMM SMOVL C00103 BC00103 V=666.7  +MOVJ EC00103
COMM SMOVL C00104 BC00104 V=166.7  +MOVJ EC00104
COMM SREFP 3 C00105 BC00105  +REFP EC00105
COMM CALL JOB:SEARCH-R1-S13D
COMM SET P062 P006
COMM SFTON3D P062
COMM SMOVL C00106 BC00106 V=166.7  +MOVJ EC00106
COMM SREFP 3 C00107 BC00107  +REFP EC00107
COMM CALL JOB:SEARCH-R1-S13D
COMM SET P062 P006
COMM SFTON3D P062
COMM SMOVL C00108 BC00108 V=250.0  +MOVJ EC00108
COMM SFTOF3D
COMM SMOVL C00109 BC00109 V=500.0  +MOVJ EC00109
COMM SMOVL C00110 BC00110 V=166.7  +MOVJ EC00110
COMM SREFP 3 C00111 BC00111  +REFP EC00111
COMM CALL JOB:SEARCH-R1-S13D
COMM SET P063 P006
COMM SFTON3D P063
COMM SMOVL C00112 BC00112 V=166.7  +MOVJ EC00112
COMM SREFP 3 C00113 BC00113  +REFP EC00113
COMM CALL JOB:SEARCH-R1-S13D
COMM SET P063 P006
COMM SFTON3D P063
COMM SMOVL C00114 BC00114 V=166.7  +MOVJ EC00114
COMM SFTOF3D
COMM SMOVL C00115 BC00115 V=1000.0  +MOVJ EC00115
COMM MOVJ C00116 BC00116 VJ=100.00  +MOVJ EC00116 VJ=30.00
COMM MOVJ C00117 BC00117 VJ=50.00  +MOVJ EC00117 VJ=30.00
COMM MOVJ C00118 BC00118 VJ=100.00  +MOVJ EC00118 VJ=100.00
COMM MOVL C00119 BC00119 V=666.7  +MOVJ EC00119 VJ=100.00
COMM SMOVL C00120 BC00120 V=166.7  +MOVJ EC00120
COMM SREFP 3 C00121 BC00121  +REFP EC00121
COMM CALL JOB:SEARCH-R1-S13D
COMM SET P023 P006
COMM SFTON3D P023
COMM SMOVL C00122 BC00122 V=166.7  +MOVJ EC00122
COMM SMOVL C00123 BC00123 V=333.3  +MOVJ EC00123
COMM SMOVL C00124 BC00124 V=166.7  +MOVJ EC00124
COMM SREFP 3 C00125 BC00125  +REFP EC00125
COMM CALL JOB:SEARCH-R1-S13D
COMM SET P023 P006
COMM SFTON3D P023
COMM SMOVL C00126 BC00126 V=166.7  +MOVJ EC00126
COMM SMOVL C00127 BC00127 V=166.7  +MOVJ EC00127
COMM SREFP 3 C00128 BC00128  +REFP EC00128
COMM CALL JOB:SEARCH-R1-S13D
COMM SET P023 P006
COMM SFTON3D P023
COMM SMOVL C00129 BC00129 V=166.7  +MOVJ EC00129
COMM MOVL C00130 BC00130 V=1000.0  +MOVJ EC00130 VJ=100.00
COMM 'EndPath S4096
COMM MOVJ C00131 BC00131 VJ=100.00  +MOVJ EC00131 VJ=100.00
COMM 'Path S4097
COMM SFTOF3D
COMM MOVJ C00132 BC00132 VJ=100.00  +MOVJ EC00132 VJ=100.00
COMM MOVL C00133 BC00133 V=666.7  +MOVJ EC00133 VJ=100.00
COMM SMOVL C00134 BC00134 V=166.7  +MOVJ EC00134
COMM SREFP 3 C00135 BC00135  +REFP EC00135
COMM CALL JOB:SEARCH-R1-S13D
COMM SET P024 P006
COMM SFTON3D P024
COMM SMOVL C00136 BC00136 V=166.7  +MOVJ EC00136
COMM SREFP 3 C00137 BC00137  +REFP EC00137
COMM CALL JOB:SEARCH-R1-S13D
COMM SET P024 P006
COMM SFTON3D P024
COMM SMOVL C00138 BC00138 V=166.7  +MOVJ EC00138
COMM SMOVL C00139 BC00139 V=166.7  +MOVJ EC00139
COMM SREFP 3 C00140 BC00140  +REFP EC00140
COMM CALL JOB:SEARCH-R1-S13D
COMM SET P024 P006
COMM SFTON3D P024
COMM SMOVL C00141 BC00141 V=166.7  +MOVJ EC00141
COMM MOVL C00142 BC00142 V=1000.0  +MOVJ EC00142 VJ=100.00
COMM 'EndPath S4097
COMM 'Path S4098
COMM SFTOF3D
COMM MOVJ C00143 BC00143 VJ=100.00  +MOVJ EC00143 VJ=100.00
COMM MOVL C00144 BC00144 V=666.7  +MOVJ EC00144 VJ=100.00
COMM SMOVL C00145 BC00145 V=166.7  +MOVJ EC00145
COMM SREFP 3 C00146 BC00146  +REFP EC00146
COMM CALL JOB:SEARCH-R1-S13D
COMM SET P035 P006
COMM SFTON3D P035
COMM SMOVL C00147 BC00147 V=166.7  +MOVJ EC00147
COMM SREFP 3 C00148 BC00148  +REFP EC00148
COMM CALL JOB:SEARCH-R1-S13D
COMM SET P035 P006
COMM SFTON3D P035
COMM SMOVL C00149 BC00149 V=166.7  +MOVJ EC00149
COMM SMOVL C00150 BC00150 V=166.7  +MOVJ EC00150
COMM SMOVL C00151 BC00151 V=166.7  +MOVJ EC00151
COMM SREFP 3 C00152 BC00152  +REFP EC00152
COMM CALL JOB:SEARCH-R1-S13D
COMM SET P035 P006
COMM SFTON3D P035
COMM SMOVL C00153 BC00153 V=166.7  +MOVJ EC00153
COMM MOVL C00154 BC00154 V=1000.0  +MOVJ EC00154 VJ=100.00
COMM 'EndPath S4098
COMM 'Path S4099
COMM SFTOF3D
COMM MOVJ C00155 BC00155 VJ=100.00  +MOVJ EC00155 VJ=100.00
COMM MOVL C00156 BC00156 V=666.7  +MOVJ EC00156 VJ=100.00
COMM SMOVL C00157 BC00157 V=166.7  +MOVJ EC00157
COMM SREFP 3 C00158 BC00158  +REFP EC00158
COMM CALL JOB:SEARCH-R1-S13D
COMM SET P029 P006
COMM SFTON3D P029
COMM SMOVL C00159 BC00159 V=166.7  +MOVJ EC00159
COMM SREFP 3 C00160 BC00160  +REFP EC00160
COMM CALL JOB:SEARCH-R1-S13D
COMM SET P029 P006
COMM SFTON3D P029
COMM SMOVL C00161 BC00161 V=166.7  +MOVJ EC00161
COMM SMOVL C00162 BC00162 V=250.0  +MOVJ EC00162
COMM SMOVL C00163 BC00163 V=166.7  +MOVJ EC00163
COMM SREFP 3 C00164 BC00164  +REFP EC00164
COMM CALL JOB:SEARCH-R1-S13D
COMM SET P029 P006
COMM SFTON3D P029
COMM SMOVL C00165 BC00165 V=166.7  +MOVJ EC00165
COMM 'EndPath S4099
COMM 'Path S4855
COMM SFTOF3D
COMM MOVL C00166 BC00166 V=666.7  +MOVJ EC00166 VJ=100.00
COMM SMOVL C00167 BC00167 V=166.7  +MOVJ EC00167
COMM SREFP 3 C00168 BC00168  +REFP EC00168
COMM CALL JOB:SEARCH-R1-S13D
COMM SET P071 P006
COMM SFTON3D P071
COMM SMOVL C00169 BC00169 V=166.7  +MOVJ EC00169
COMM SREFP 3 C00170 BC00170  +REFP EC00170
COMM CALL JOB:SEARCH-R1-S13D
COMM SET P071 P006
COMM SFTON3D P071
COMM SMOVL C00171 BC00171 V=166.7  +MOVJ EC00171
COMM SMOVL C00172 BC00172 V=166.7  +MOVJ EC00172
COMM SREFP 3 C00173 BC00173  +REFP EC00173
COMM CALL JOB:SEARCH-R1-S13D
COMM SET P071 P006
COMM SFTON3D P071
COMM SMOVL C00174 BC00174 V=166.7  +MOVJ EC00174
COMM MOVL C00175 BC00175 V=1000.0  +MOVJ EC00175 VJ=100.00
COMM 'EndPath S4855
COMM 'Path S4856
COMM SFTOF3D
COMM MOVJ C00176 BC00176 VJ=100.00  +MOVJ EC00176 VJ=100.00
COMM MOVL C00177 BC00177 V=666.7  +MOVJ EC00177 VJ=100.00
COMM SMOVL C00178 BC00178 V=166.7  +MOVJ EC00178
COMM SREFP 3 C00179 BC00179  +REFP EC00179
COMM CALL JOB:SEARCH-R1-S13D
COMM SET P072 P006
COMM SFTON3D P072
COMM SMOVL C00180 BC00180 V=166.7  +MOVJ EC00180
COMM SREFP 3 C00181 BC00181  +REFP EC00181
COMM CALL JOB:SEARCH-R1-S13D
COMM SET P072 P006
COMM SFTON3D P072
COMM SMOVL C00182 BC00182 V=166.7  +MOVJ EC00182
COMM MOVL C00183 BC00183 V=1000.0  +MOVJ EC00183 VJ=100.00
COMM 'EndPath S4856
COMM MOVJ C00184 BC00184 VJ=100.00  +MOVJ EC00184 VJ=100.00
COMM 'Path S4857
COMM SFTOF3D
COMM MOVJ C00185 BC00185 VJ=100.00  +MOVJ EC00185 VJ=100.00
COMM MOVL C00186 BC00186 V=666.7  +MOVJ EC00186 VJ=100.00
COMM SMOVL C00187 BC00187 V=166.7  +MOVJ EC00187
COMM SREFP 3 C00188 BC00188  +REFP EC00188
COMM CALL JOB:SEARCH-R1-S13D
COMM SET P073 P006
COMM SFTON3D P073
COMM SMOVL C00189 BC00189 V=166.7  +MOVJ EC00189
COMM SMOVL C00190 BC00190 V=166.7  +MOVJ EC00190
COMM SREFP 3 C00191 BC00191  +REFP EC00191
COMM CALL JOB:SEARCH-R1-S13D
COMM SET P073 P006
COMM SFTON3D P073
COMM SMOVL C00192 BC00192 V=166.7  +MOVJ EC00192
COMM SMOVL C00193 BC00193 V=166.7  +MOVJ EC00193
COMM SREFP 3 C00194 BC00194  +REFP EC00194
COMM CALL JOB:SEARCH-R1-S13D
COMM SET P073 P006
COMM SFTON3D P073
COMM SMOVL C00195 BC00195 V=166.7  +MOVJ EC00195
COMM MOVL C00196 BC00196 V=1000.0  +MOVJ EC00196 VJ=100.00
COMM 'EndPath S4857
COMM MOVJ C00197 BC00197 VJ=100.00  +MOVJ EC00197 VJ=100.00
COMM 'Path S4858
COMM SFTOF3D
COMM MOVJ C00198 BC00198 VJ=100.00  +MOVJ EC00198 VJ=100.00
COMM MOVL C00199 BC00199 V=666.7  +MOVJ EC00199 VJ=100.00
COMM SMOVL C00200 BC00200 V=166.7  +MOVJ EC00200
COMM SREFP 3 C00201 BC00201  +REFP EC00201
COMM CALL JOB:SEARCH-R1-S13D
COMM SET P074 P006
COMM SFTON3D P074
COMM SMOVL C00202 BC00202 V=166.7  +MOVJ EC00202
COMM SREFP 3 C00203 BC00203  +REFP EC00203
COMM CALL JOB:SEARCH-R1-S13D
COMM SET P074 P006
COMM SFTON3D P074
COMM SMOVL C00204 BC00204 V=166.7  +MOVJ EC00204
COMM MOVL C00205 BC00205 V=1000.0  +MOVJ EC00205 VJ=100.00
COMM 'EndPath S4858
COMM MOVJ C00206 BC00206 VJ=100.00  +MOVJ EC00206 VJ=100.00
COMM MOVJ C00207 BC00207 VJ=100.00  +MOVJ EC00207 VJ=100.00
COMM 'Path S4100
COMM SFTOF3D
COMM MOVJ C00208 BC00208 VJ=100.00  +MOVJ EC00208 VJ=100.00
COMM MOVL C00209 BC00209 V=666.7  +MOVJ EC00209 VJ=100.00
COMM SMOVL C00210 BC00210 V=166.7  +MOVJ EC00210
COMM SREFP 3 C00211 BC00211  +REFP EC00211
COMM CALL JOB:SEARCH-R1-S13D
COMM SET P026 P006
COMM SFTON3D P026
COMM SMOVL C00212 BC00212 V=166.7  +MOVJ EC00212
COMM SREFP 3 C00213 BC00213  +REFP EC00213
COMM CALL JOB:SEARCH-R1-S13D
COMM SET P026 P006
COMM SFTON3D P026
COMM SMOVL C00214 BC00214 V=166.7  +MOVJ EC00214
COMM SMOVL C00215 BC00215 V=666.7  +MOVJ EC00215
COMM SMOVL C00216 BC00216 V=666.7  +MOVJ EC00216
COMM SMOVL C00217 BC00217 V=666.7  +MOVJ EC00217
COMM SMOVL C00218 BC00218 V=166.7  +MOVJ EC00218
COMM SREFP 3 C00219 BC00219  +REFP EC00219
COMM CALL JOB:SEARCH-R1-S13D
COMM SET P026 P006
COMM SFTON3D P026
COMM SMOVL C00220 BC00220 V=250.0  +MOVJ EC00220
COMM SMOVL C00221 BC00221 V=666.7  +MOVJ EC00221
COMM MOVL C00222 BC00222 V=1000.0  +MOVJ EC00222 VJ=100.00
COMM 'EndPath S4100
COMM MOVJ C00223 BC00223 VJ=50.00  +MOVJ EC00223 VJ=100.00
COMM 'Path S4101
COMM SFTOF3D
COMM MOVJ C00224 BC00224 VJ=50.00  +MOVJ EC00224 VJ=100.00
COMM MOVL C00225 BC00225 V=666.7  +MOVJ EC00225 VJ=100.00
COMM SMOVL C00226 BC00226 V=166.7  +MOVJ EC00226
COMM SREFP 3 C00227 BC00227  +REFP EC00227
COMM CALL JOB:SEARCH-R1-S13D
COMM SET P025 P006
COMM SFTON3D P025
COMM SMOVL C00228 BC00228 V=166.7  +MOVJ EC00228
COMM SREFP 3 C00229 BC00229  +REFP EC00229
COMM CALL JOB:SEARCH-R1-S13D
COMM SET P025 P006
COMM SFTON3D P025
COMM SMOVL C00230 BC00230 V=166.7  +MOVJ EC00230
COMM SMOVL C00231 BC00231 V=333.3  +MOVJ EC00231
COMM SMOVL C00232 BC00232 V=166.7  +MOVJ EC00232
COMM SREFP 3 C00233 BC00233  +REFP EC00233
COMM CALL JOB:SEARCH-R1-S13D
COMM SET P025 P006
COMM SFTON3D P025
COMM SMOVL C00234 BC00234 V=166.7  +MOVJ EC00234
COMM MOVL C00235 BC00235 V=1000.0  +MOVJ EC00235 VJ=100.00
COMM 'EndPath S4101
COMM MOVJ C00236 BC00236 VJ=100.00  +MOVJ EC00236 VJ=100.00
COMM 'Path S4102
COMM SFTOF3D
COMM MOVJ C00237 BC00237 VJ=100.00  +MOVJ EC00237 VJ=100.00
COMM MOVL C00238 BC00238 V=666.7  +MOVJ EC00238 VJ=100.00
COMM SMOVL C00239 BC00239 V=166.7  +MOVJ EC00239
COMM SREFP 3 C00240 BC00240  +REFP EC00240
COMM CALL JOB:SEARCH-R1-S13D
COMM SET P028 P006
COMM SFTON3D P028
COMM SMOVL C00241 BC00241 V=166.7  +MOVJ EC00241
COMM SREFP 3 C00242 BC00242  +REFP EC00242
COMM CALL JOB:SEARCH-R1-S13D
COMM SET P028 P006
COMM SFTON3D P028
COMM SMOVL C00243 BC00243 V=166.7  +MOVJ EC00243
COMM SMOVL C00244 BC00244 V=333.3  +MOVJ EC00244
COMM SMOVL C00245 BC00245 V=166.7  +MOVJ EC00245
COMM SREFP 3 C00246 BC00246  +REFP EC00246
COMM CALL JOB:SEARCH-R1-S13D
COMM SET P028 P006
COMM SFTON3D P028
COMM SMOVL C00247 BC00247 V=166.7  +MOVJ EC00247
COMM MOVL C00248 BC00248 V=1000.0  +MOVJ EC00248 VJ=100.00
COMM 'EndPath S4102
COMM MOVJ C00249 BC00249 VJ=100.00  +MOVJ EC00249 VJ=100.00
COMM 'Path S4103
COMM SFTOF3D
COMM MOVJ C00250 BC00250 VJ=100.00  +MOVJ EC00250 VJ=100.00
COMM MOVL C00251 BC00251 V=666.7  +MOVJ EC00251 VJ=100.00
COMM SMOVL C00252 BC00252 V=166.7  +MOVJ EC00252
COMM SREFP 3 C00253 BC00253  +REFP EC00253
COMM CALL JOB:SEARCH-R1-S13D
COMM SET P033 P006
COMM SFTON3D P033
COMM SMOVL C00254 BC00254 V=166.7  +MOVJ EC00254
COMM SMOVL C00255 BC00255 V=166.7  +MOVJ EC00255
COMM SREFP 3 C00256 BC00256  +REFP EC00256
COMM CALL JOB:SEARCH-R1-S13D
COMM SET P033 P006
COMM SFTON3D P033
COMM SMOVL C00257 BC00257 V=166.7  +MOVJ EC00257
COMM SMOVL C00258 BC00258 V=166.7  +MOVJ EC00258
COMM SMOVL C00259 BC00259 V=166.7  +MOVJ EC00259
COMM SREFP 3 C00260 BC00260  +REFP EC00260
COMM CALL JOB:SEARCH-R1-S13D
COMM SET P033 P006
COMM SFTON3D P033
COMM SMOVL C00261 BC00261 V=166.7  +MOVJ EC00261
COMM MOVL C00262 BC00262 V=1000.0  +MOVJ EC00262 VJ=100.00
COMM 'EndPath S4103
COMM 'Path S4104
COMM SFTOF3D
COMM MOVJ C00263 BC00263 VJ=100.00  +MOVJ EC00263 VJ=100.00
COMM MOVL C00264 BC00264 V=666.7  +MOVJ EC00264 VJ=100.00
COMM SMOVL C00265 BC00265 V=166.7  +MOVJ EC00265
COMM SREFP 3 C00266 BC00266  +REFP EC00266
COMM CALL JOB:SEARCH-R1-S13D
COMM SET P027 P006
COMM SFTON3D P027
COMM SMOVL C00267 BC00267 V=250.0  +MOVJ EC00267
COMM SMOVL C00268 BC00268 V=166.7  +MOVJ EC00268
COMM SREFP 3 C00269 BC00269  +REFP EC00269
COMM CALL JOB:SEARCH-R1-S13D
COMM SET P027 P006
COMM SFTON3D P027
COMM SMOVL C00270 BC00270 V=166.7  +MOVJ EC00270
COMM SMOVL C00271 BC00271 V=166.7  +MOVJ EC00271
COMM SREFP 3 C00272 BC00272  +REFP EC00272
COMM CALL JOB:SEARCH-R1-S13D
COMM SET P027 P006
COMM SFTON3D P027
COMM SMOVL C00273 BC00273 V=166.7  +MOVJ EC00273
COMM MOVL C00274 BC00274 V=1000.0  +MOVJ EC00274 VJ=100.00
COMM 'EndPath S4104
COMM MOVJ C00275 BC00275 VJ=100.00  +MOVJ EC00275 VJ=100.00
COMM 'Path S4105
COMM SFTOF3D
COMM MOVJ C00276 BC00276 VJ=100.00  +MOVJ EC00276 VJ=100.00
COMM MOVL C00277 BC00277 V=666.7  +MOVJ EC00277 VJ=100.00
COMM SMOVL C00278 BC00278 V=166.7  +MOVJ EC00278
COMM SREFP 3 C00279 BC00279  +REFP EC00279
COMM CALL JOB:SEARCH-R1-S13D
COMM SET P030 P006
COMM SFTON3D P030
COMM SMOVL C00280 BC00280 V=166.7  +MOVJ EC00280
COMM SREFP 3 C00281 BC00281  +REFP EC00281
COMM CALL JOB:SEARCH-R1-S13D
COMM SET P030 P006
COMM SFTON3D P030
COMM SMOVL C00282 BC00282 V=166.7  +MOVJ EC00282
COMM MOVL C00283 BC00283 V=1000.0  +MOVJ EC00283 VJ=100.00
COMM 'EndPath S4105
COMM 'Path S4106
COMM SFTOF3D
COMM MOVJ C00284 BC00284 VJ=100.00  +MOVJ EC00284 VJ=100.00
COMM MOVL C00285 BC00285 V=666.7  +MOVJ EC00285 VJ=100.00
COMM SMOVL C00286 BC00286 V=166.7  +MOVJ EC00286
COMM SREFP 3 C00287 BC00287  +REFP EC00287
COMM CALL JOB:SEARCH-R1-S13D
COMM SET P031 P006
COMM SFTON3D P031
COMM SMOVL C00288 BC00288 V=166.7  +MOVJ EC00288
COMM SREFP 3 C00289 BC00289  +REFP EC00289
COMM CALL JOB:SEARCH-R1-S13D
COMM SET P031 P006
COMM SFTON3D P031
COMM SMOVL C00290 BC00290 V=166.7  +MOVJ EC00290
COMM MOVL C00291 BC00291 V=1000.0  +MOVJ EC00291 VJ=100.00
COMM 'EndPath S4106
COMM MOVJ C00292 BC00292 VJ=100.00  +MOVJ EC00292 VJ=100.00
COMM 'Path S4107
COMM SFTOF3D
COMM MOVJ C00293 BC00293 VJ=100.00  +MOVJ EC00293 VJ=100.00
COMM MOVL C00294 BC00294 V=666.7  +MOVJ EC00294 VJ=100.00
COMM SMOVL C00295 BC00295 V=166.7  +MOVJ EC00295
